(* CODESYS project Project1.project

Project tree, tasks and I/O mapping:
  PLC_AC500_V3 : PM5032-T-ETH, ABB AG, order no. 1SAP123400R0x72, version 3.7.0.0
    application Application
      task Task (cyclic, interval t#10ms, priority 14, watchdog t#20ms x 1) calls batching8, batching7
      task VISU_TASK (cyclic, interval 100 ms, priority 16) calls VisuElems.Visu_Prg
      CheckConfigurationObject
      program PLC_PRG [ST]
      program batching1 [ST]
      Diagnosis/
        text list Diag_IO_Bus
        text list Diag_V3_PLC
      program batching2 [ST]
      program batching3 [ST]
      program batching4 [ST]
      visualisation batching4_vis
      program batching5 [ST]
      global variables GVL
      function block Auto_Batching [ST]
      function block Manual_Batching [ST]
      program batching6 [ST]
      function block Auto_Batching_V7 [ST]
      function block Manual_Batching_V7 [ST]
      program batching7 [ST]
      function block Auto_Batching_V8 [ST]
      function block Manual_Batching_V8 [ST]
      program batching8 [ST]
      function block Auto_Batching_V9 [ST]
      function block Manual_Batching_V9 [ST]
      program batching9 [ST]
    OnBoard_IO : 12DI/8DO-T/2DC, ABB AG, version 3.7.0.0
        unmapped channels: Fast inputs DI0-DI3, Fast inputs DI4-DI7, Standard inputs DI8-DI11, Digital inputs - Transistor, Fast outputs DO0-DO3, Fast outputs DO4-DO7, Digital outputs - Transistor
    IO_Bus : I/O-Bus, ABB AG, version 3.7.0.0
    Interfaces : Interfaces, ABB AG, version 3.7.0.0
      OptionSlot_1
      OptionSlot_2
      Ethernet : Ethernet, ABB AG, version 3.7.0.0
        ETH1 : IP Settings, ABB AG, version 3.7.0.0
          NetConfig : NetConfig, ABB AG, version 3.7.0.0
        Protocols : Client Protocols, ABB AG, version 3.7.0.0
    OnBoard_RTC : OnBoard RTC, ABB AG, version 3.7.0.0
  text list GlobalTextList
*)

// PLC_AC500_V3/Application/GVL
{attribute 'qualified_only'}
VAR_GLOBAL
    Recipe_Weights : ARRAY[1..20] OF REAL := [
        50.0,   // Mat 1 (Auto Silo 1)
        15.0,   // Mat 2 (Auto Silo 2)
        28.0,   // Mat 3
        31.0,   // Mat 4 (Auto Silo 4)
        150.0,  // Mat 5 (Auto Silo 5)
        10.0,   // Mat 6 (Auto Silo 6)
        12.0,   // Mat 7 (Manual Silo 7)
        8.0,    // Mat 8 (Manual Silo 8)
        25.0,   // Mat 9 (Manual Silo 9)
        5.0,    // Mat 10 (Manual Silo 10)
        18.0,   // Mat 11 (Manual Silo 11)
        22.0,   // Mat 12 (Manual Silo 12)
        30.0,   // Mat 13 (Manual Silo 13)
        14.0,   // Mat 14 (Manual Silo 14)
        9.0,    // Mat 15 (Manual Silo 15)
        11.0,   // Mat 16 (Manual Silo 16)
        0.0, 0.0, 0.0, 0.0
    ];
END_VAR

// PLC_AC500_V3/Application/batching8
PROGRAM batching8
VAR
    Auto_Ctrl : Auto_Batching_V8;
    Manual_Ctrl : Manual_Batching_V8;
    
    (* Global Inputs & Toggles *)
    Start_Button : BOOL;
    E_Stop_Active : BOOL;
    
    (* Parallel Weight Feedbacks *)
    load_cell_auto : REAL;
    load_cell_manual : REAL;
    
    (* Sub-Block Diagnostic Indicators - Ordered exactly below loadcell *)
    Auto_Active_Mat : INT;
    Auto_Active_Bin : INT;
    Auto_Active_Target : REAL; // Active Target Weight for Auto (displays GVL setpoint)
    Auto_Err : INT;
    Auto_Msg : STRING;
    
    Manual_Active_Mat : INT;
    Manual_Active_Bin : INT;
    Manual_Active_Target : REAL; // Active Target Weight for Manual (displays GVL setpoint)
    Manual_Err : INT;
    Manual_Msg : STRING;
    
    (* Process Outputs *)
    Auto_Bin : ARRAY[1..6] OF BOOL; // Valve control outputs (Coarse)
    auto_bin_cutoff : ARRAY[1..6] OF BOOL; // Cutoff indicators (Fine)
    auto_bin_motor : ARRAY[1..6] OF BOOL; // Conveyor/feeder motor outputs
    
    Manual_Bin : ARRAY[1..10] OF BOOL; // Prompt indicators (Coarse)
    manual_bin_cutoff : ARRAY[1..10] OF BOOL; // Cutoff indicators (Fine)
    manual_bin_motor : ARRAY[1..10] OF BOOL; // Conveyor/feeder motor outputs
    
    Auto_Weights : ARRAY[1..6] OF REAL;
    Manual_Weights : ARRAY[1..10] OF REAL;
    
    Auto_Complete : BOOL;
    Manual_Complete : BOOL;
    Sequence_Complete : BOOL;
    
    (* Diagnostics & Interlocks *)
    Error_Code : INT := 0;
    Status_Message : STRING := 'System Ready';
    
    (* Array Configurations & Mapping - Renamed for clarity *)
    Auto_Bin_Material_Mapping : ARRAY[1..6] OF INT := [1, 2, 0, 4, 5, 6];
    Manual_Bin_Material_Mapping : ARRAY[1..10] OF INT := [7, 8, 0, 10, 11, 12, 13, 14, 15, 16];
    Auto_Bin_Cutoff_Weights : ARRAY[1..6] OF REAL := [2.0, 1.5, 0.0, 3.0, 5.0, 1.0]; // Cutoff margins (kg)
    Manual_Bin_Cutoff_Weights : ARRAY[1..10] OF REAL := [2.0, 1.5, 0.0, 3.0, 5.0, 1.0, 2.0, 2.0, 2.0, 2.0];
    
    i : INT;
    j : INT;
    Duplicate_Found : BOOL;
    Invalid_Material_Range : BOOL;
    Zero_Target_Found : BOOL;
    Conf_Err_Id : INT;
END_VAR

(* 1. STARTUP CONFIGURATION CHECKS *)
Duplicate_Found := FALSE;
Invalid_Material_Range := FALSE;
Zero_Target_Found := FALSE;

FOR i := 1 TO 6 DO
    (* Check 2: Out of Range (Auto) *)
    IF Auto_Bin_Material_Mapping[i] < 0 OR Auto_Bin_Material_Mapping[i] > 20 THEN
        Invalid_Material_Range := TRUE;
    END_IF;
    
    (* Check 3: Zero Target (Auto) *)
    IF Auto_Bin_Material_Mapping[i] <> 0 AND Auto_Bin_Material_Mapping[i] <= 20 THEN
        IF GVL.Recipe_Weights[Auto_Bin_Material_Mapping[i]] = 0.0 THEN
            Zero_Target_Found := TRUE;
        END_IF;
    END_IF;
    
    (* Check 1: Duplicate Cross-Array Material ID *)
    IF Auto_Bin_Material_Mapping[i] <> 0 AND Auto_Bin_Material_Mapping[i] <= 20 THEN
        FOR j := 1 TO 10 DO
            IF Auto_Bin_Material_Mapping[i] = Manual_Bin_Material_Mapping[j] THEN
                Duplicate_Found := TRUE;
            END_IF;
        END_FOR;
    END_IF;
END_FOR;

FOR j := 1 TO 10 DO
    (* Check 2: Out of Range (Manual) *)
    IF Manual_Bin_Material_Mapping[j] < 0 OR Manual_Bin_Material_Mapping[j] > 20 THEN
        Invalid_Material_Range := TRUE;
    END_IF;
    
    (* Check 3: Zero Target (Manual) *)
    IF Manual_Bin_Material_Mapping[j] <> 0 AND Manual_Bin_Material_Mapping[j] <= 20 THEN
        IF GVL.Recipe_Weights[Manual_Bin_Material_Mapping[j]] = 0.0 THEN
            Zero_Target_Found := TRUE;
        END_IF;
    END_IF;
END_FOR;

(* Configuration Error Resolution *)
IF Duplicate_Found THEN
    Error_Code := 1;
    Status_Message := 'Error 1: Duplicate Material ID mapped in Auto and Manual!';
ELSIF Invalid_Material_Range THEN
    Error_Code := 2;
    Status_Message := 'Error 2: Material Index configuration out of range (1..20)!';
ELSIF Zero_Target_Found THEN
    Error_Code := 3;
    Status_Message := 'Error 3: Configured Material ID has a 0.0 kg target weight!';
ELSE
    IF Error_Code <= 3 THEN
        Error_Code := 0;
    END_IF;
END_IF;

(* Abort sequences if a configuration error exists *)
IF Error_Code >= 1 AND Error_Code <= 3 THEN
    FOR i := 1 TO 6 DO Auto_Bin[i] := FALSE; auto_bin_cutoff[i] := FALSE; auto_bin_motor[i] := FALSE; END_FOR;
    FOR i := 1 TO 10 DO Manual_Bin[i] := FALSE; manual_bin_cutoff[i] := FALSE; manual_bin_motor[i] := FALSE; END_FOR;
    Auto_Ctrl(Start_Button := FALSE, E_Stop_Active := TRUE, load_cell_value := load_cell_auto);
    Manual_Ctrl(Start_Button := FALSE, E_Stop_Active := TRUE, load_cell_value := load_cell_manual);
    Auto_Active_Target := 0.0;
    Manual_Active_Target := 0.0;
    RETURN;
END_IF;


(* 2. CONCURRENT EXECUTION OF FB INSTANCES *)
Auto_Ctrl(
    Start_Button := Start_Button,
    E_Stop_Active := E_Stop_Active,
    load_cell_value := load_cell_auto,
    Auto_Bin_Material_Mapping := Auto_Bin_Material_Mapping,
    Auto_Bin_Cutoff_Weights := Auto_Bin_Cutoff_Weights,
    Auto_Bin => Auto_Bin,
    auto_bin_cutoff => auto_bin_cutoff,
    auto_bin_motor => auto_bin_motor,
    Actual_Weights => Auto_Weights,
    Sequence_Complete => Auto_Complete,
    Active_Material_ID => Auto_Active_Mat,
    Active_Bin_ID => Auto_Active_Bin,
    Active_Target_Weight => Auto_Active_Target,
    Error_Code => Auto_Err,
    Status_Message => Auto_Msg
);

Manual_Ctrl(
    Start_Button := Start_Button,
    E_Stop_Active := E_Stop_Active,
    load_cell_value := load_cell_manual,
    Manual_Bin_Material_Mapping := Manual_Bin_Material_Mapping,
    Manual_Bin_Cutoff_Weights := Manual_Bin_Cutoff_Weights,
    Manual_Bin => Manual_Bin,
    manual_bin_cutoff => manual_bin_cutoff,
    manual_bin_motor => manual_bin_motor,
    Actual_Weights => Manual_Weights,
    Sequence_Complete => Manual_Complete,
    Active_Material_ID => Manual_Active_Mat,
    Active_Bin_ID => Manual_Active_Bin,
    Active_Target_Weight => Manual_Active_Target,
    Error_Code => Manual_Err,
    Status_Message => Manual_Msg
);

(* Runtime Error Mapping & Aggregation *)
IF Auto_Err <> 0 THEN
    Error_Code := Auto_Err;
    Status_Message := CONCAT('Auto Error: ', Auto_Msg);
ELSIF Manual_Err <> 0 THEN
    Error_Code := Manual_Err;
    Status_Message := CONCAT('Manual Error: ', Manual_Msg);
ELSE
    Error_Code := 0;
    
    Sequence_Complete := Auto_Complete AND Manual_Complete;
    IF Sequence_Complete THEN
        Status_Message := 'Batch Sequence Completed';
    ELSIF Start_Button THEN
        Status_Message := 'Batch Sequence Running';
    ELSE
        Status_Message := 'System Ready';
    END_IF;
END_IF;

END_PROGRAM

// PLC_AC500_V3/Application/Auto_Batching_V8
FUNCTION_BLOCK Auto_Batching_V8
VAR_INPUT
    Start_Button : BOOL;      // Signal to start the batching sequence
    E_Stop_Active : BOOL;     // Emergency Stop active signal
    Discharge_Bin_Feedback : ARRAY[1..6] OF BOOL; // Physical valve feedbacks
    Auto_Bin_Material_Mapping : ARRAY[1..6] OF INT; // Material index mapping for 6 bins
    Auto_Bin_Cutoff_Weights : ARRAY[1..6] OF REAL; // Cutoff weight thresholds (kg)
END_VAR
VAR_IN_OUT
    load_cell_value : REAL;   // Weight value read/written from load cell
END_VAR
VAR_OUTPUT
    Auto_Bin : ARRAY[1..6] OF BOOL; // Coarse feed valve outputs
    auto_bin_cutoff : ARRAY[1..6] OF BOOL; // Fine feed cutoff trigger indicators
    auto_bin_motor : ARRAY[1..6] OF BOOL; // Main conveyor motor outputs
    Actual_Weights : ARRAY[1..6] OF REAL; // Actual weight poured per silo
    Sequence_Complete : BOOL;  // Batch complete flag
    Active_Material_ID : INT;  // Currently active ingredient ID
    Active_Bin_ID : INT;       // Currently active physical Bin ID (1..6)
    Active_Target_Weight : REAL; // Recipe target weight of active bin
    Error_Code : INT;          // Active error code
    Status_Message : STRING;   // Diagnostic text message
END_VAR
VAR
    Step : INT := 0;          // State machine index (0: Idle, 1..6: Bins, 11..16: Delays, 7: Settling, 8: Complete, 99: Error)
    bin_last_weight : REAL;   // Baseline weight on the load cell before starting current bin
    actual_bin : REAL;        // Current weight added from active bin
    target_act_bin : REAL;    // Target weight to add from the active bin
    bin_set_value : REAL;     // Setpoint weight for current active step
    cutoff_trigger_weight : REAL; // Calculated target threshold weight minus cutoff value
    
    Mat_Idx : INT;
    i : INT;                  // General loop index
    
    (* TIMERS FOR TRANSITIONS & DELAYS *)
    Transition_Timer : TON;
    Completion_Timer : TON;
    Step_Delay_Time : TIME := T#2S;
    Post_Complete_Delay : TIME := T#2S;
    
    (* SELF-CONTAINED SIMULATION VARIABLES *)
    Simulation_Mode : BOOL := TRUE;
    Sim_Rate : REAL := 10.0;            // Simulated pouring speed (10.0 kg/s)
    Sim_Timer : TON;
    Start_Sim_Weight : REAL;
    Discharge_Active : BOOL;
END_VAR

(* Auto Batching FB V8 matching batching7 sequence exactly *)

(* 1. SELF-CONTAINED SIMULATION WEIGHT MANAGEMENT *)
IF Simulation_Mode AND Step <> 99 THEN
    (* Reset simulation to baseline *)
    IF Step = 0 AND NOT Start_Button AND NOT Sequence_Complete THEN
        load_cell_value := 0.0;
        bin_last_weight := 0.0;
        Start_Sim_Weight := 0.0;
        Sim_Timer(IN := FALSE);
    END_IF;
    
    (* Check if any valve is actively discharging *)
    Discharge_Active := FALSE;
    IF Step >= 1 AND Step <= 6 THEN
        Discharge_Active := auto_bin_motor[Step];
    END_IF;
    
    (* Simulate weight gain on the load cell *)
    IF Discharge_Active THEN
        Sim_Timer(IN := TRUE, PT := T#1000S);
        load_cell_value := Start_Sim_Weight + (TIME_TO_REAL(Sim_Timer.ET) / 1000.0) * Sim_Rate;
    ELSE
        Sim_Timer(IN := FALSE);
        Start_Sim_Weight := load_cell_value;
    END_IF;
END_IF;


(* 2. EMERGENCY STOP LOGIC (Error 12) *)
IF E_Stop_Active THEN
    FOR i := 1 TO 6 DO
        Auto_Bin[i] := FALSE;
        auto_bin_cutoff[i] := FALSE;
        auto_bin_motor[i] := FALSE;
    END_FOR;
    Sequence_Complete := FALSE;
    Active_Material_ID := 0;
    Active_Bin_ID := 0;
    Active_Target_Weight := 0.0;
    Error_Code := 12;
    Status_Message := 'Error 12: Emergency Stop Active!';
    Step := 99;
    Transition_Timer(IN := FALSE);
    Completion_Timer(IN := FALSE);
    RETURN;
END_IF;


(* 3. RECIPE SEQUENCE START *)
IF Step = 0 AND Start_Button THEN
    Step := 1;
    bin_last_weight := load_cell_value;
    Sequence_Complete := FALSE;
    Error_Code := 0;
    Status_Message := 'Auto Batch Started';
    Active_Target_Weight := 0.0;
    (* Clear actual weights and outputs on start *)
    FOR i := 1 TO 6 DO
        Actual_Weights[i] := 0.0;
        Auto_Bin[i] := FALSE;
        auto_bin_cutoff[i] := FALSE;
        auto_bin_motor[i] := FALSE;
    END_FOR;
END_IF;


(* 4. SEQUENCE CONTROL STATE MACHINE *)
CASE Step OF
    0:
        Active_Material_ID := 0;
        Active_Bin_ID := 0;
        Active_Target_Weight := 0.0;
        IF Error_Code = 0 THEN Status_Message := 'Auto Idle'; END_IF;
        
    1..6: (* Discharging Silos 1 to 6 *)
        Mat_Idx := Auto_Bin_Material_Mapping[Step];
        
        IF Mat_Idx = 0 THEN
            (* Skip this bin instantly *)
            Step := Step + 1;
        ELSE
            (* Fetch target weight from global Recipe_Weights array *)
            bin_set_value := GVL.Recipe_Weights[Mat_Idx];
            target_act_bin := bin_set_value;
            Active_Target_Weight := target_act_bin;
            
            (* Calculate weight added by current active bin *)
            actual_bin := load_cell_value - bin_last_weight;
            Actual_Weights[Step] := actual_bin;
            
            (* Get cutoff threshold *)
            cutoff_trigger_weight := target_act_bin - Auto_Bin_Cutoff_Weights[Step];
            
            Active_Material_ID := Mat_Idx;
            Active_Bin_ID := Step;
            Status_Message := 'Auto Pouring';
            
            (* COARSE/FINE FEED TRANSITIONS *)
            IF actual_bin < cutoff_trigger_weight THEN
                (* Phase 1: Coarse Feed (Conveyor Motor ON, Main Valve ON, Fine Cutoff OFF) *)
                Auto_Bin[Step] := TRUE;
                auto_bin_cutoff[Step] := FALSE;
                auto_bin_motor[Step] := TRUE;
            ELSIF actual_bin < target_act_bin THEN
                (* Phase 2: Fine Feed (Conveyor Motor ON, Main Valve OFF, Fine Cutoff ON) *)
                Auto_Bin[Step] := FALSE;
                auto_bin_cutoff[Step] := TRUE;
                auto_bin_motor[Step] := TRUE;
            ELSE
                (* Phase 3: Completed (All OFF) *)
                Auto_Bin[Step] := FALSE;
                auto_bin_cutoff[Step] := FALSE;
                auto_bin_motor[Step] := FALSE;
                bin_last_weight := load_cell_value;
                Active_Target_Weight := 0.0;
                Step := 10 + Step; // Offset to separate transition states
            END_IF;
            
            (* RUNTIME CHECKS *)
            (* Check 21 & 22: Scale Limits *)
            IF load_cell_value > 500.0 THEN
                Error_Code := 21;
                Status_Message := 'Error 21: Scale Overloaded!';
                Step := 99;
                RETURN;
            ELSIF load_cell_value < 0.0 THEN
                Error_Code := 22;
                Status_Message := 'Error 22: Scale Underloaded/Fault!';
                Step := 99;
                RETURN;
            END_IF;
        END_IF;

    11..15: (* Transition Delays (Between Bins) *)
        Active_Material_ID := 0;
        Active_Bin_ID := 0;
        Active_Target_Weight := 0.0;
        Status_Message := 'Transition Delay';
        
        Transition_Timer(IN := TRUE, PT := Step_Delay_Time);
        IF Transition_Timer.Q THEN
            Transition_Timer(IN := FALSE);
            Step := (Step - 10) + 1; // Advance to next bin
        END_IF;
        
    16: (* Transition Delay After Last Bin (Bin 6) Closes *)
        Active_Material_ID := 0;
        Active_Bin_ID := 0;
        Active_Target_Weight := 0.0;
        Status_Message := 'Settling Last Bin';
        
        Transition_Timer(IN := TRUE, PT := Step_Delay_Time);
        IF Transition_Timer.Q THEN
            Transition_Timer(IN := FALSE);
            Step := 7; // Go to post-discharge wait step
        END_IF;

    7: (* Wait 2 Seconds After Closing the Last Bin *)
        Active_Material_ID := 0;
        Active_Bin_ID := 0;
        Active_Target_Weight := 0.0;
        Status_Message := 'Settling Delay';
        Completion_Timer(IN := TRUE, PT := Post_Complete_Delay);
        IF Completion_Timer.Q THEN
            Completion_Timer(IN := FALSE);
            Step := 8; // Proceed to reset last weight
        END_IF;
        
    8: (* Reset bin_last_weight to 0 & Complete *)
        Active_Material_ID := 0;
        Active_Bin_ID := 0;
        Active_Target_Weight := 0.0;
        Status_Message := 'Sequence Completed';
        bin_last_weight := 0.0;
        Sequence_Complete := TRUE;
        
        IF NOT Start_Button THEN
            Step := 0;
            Sequence_Complete := FALSE;
            (* Reset all actual weights at completion once start is released *)
            FOR i := 1 TO 6 DO
                Actual_Weights[i] := 0.0;
            END_FOR;
        END_IF;
        
    99: (* Error Abort state *)
        FOR i := 1 TO 6 DO 
            Auto_Bin[i] := FALSE; 
            auto_bin_cutoff[i] := FALSE;
            auto_bin_motor[i] := FALSE;
        END_FOR;
        Active_Material_ID := 0;
        Active_Bin_ID := 0;
        Active_Target_Weight := 0.0;
        IF NOT Start_Button THEN
            Step := 0;
            Error_Code := 0;
            Status_Message := 'Auto Idle';
        END_IF;
END_CASE;

END_FUNCTION_BLOCK

// PLC_AC500_V3/Application/batching7
PROGRAM batching7
VAR
    Auto_Ctrl : Auto_Batching_V7;
    Manual_Ctrl : Manual_Batching_V7;
    
    (* Global Inputs & Toggles *)
    Start_Button : BOOL;
    E_Stop_Active : BOOL;
    
    (* Parallel Weight Feedbacks *)
    load_cell_auto : REAL;
    load_cell_manual : REAL;
    
    (* Process Outputs *)
    Auto_Bin : ARRAY[1..6] OF BOOL;
    Manual_Bin : ARRAY[1..10] OF BOOL;
    
    Auto_Weights : ARRAY[1..6] OF REAL;
    Manual_Weights : ARRAY[1..10] OF REAL;
    
    Auto_Complete : BOOL;
    Manual_Complete : BOOL;
    Sequence_Complete : BOOL;
    
    (* Cross-Validation *)
    Error_Code : INT := 0; // 0 = OK, 1 = Duplicate Material ID detected
    Status_Message : STRING := 'System Ready';
    
    (* Arrays defined here to allow check before FB execution *)
    Bin_Material_Index : ARRAY[1..6] OF INT := [1, 2, 0, 4, 5, 6];
    Bin_Manual_Index : ARRAY[1..10] OF INT := [7, 8, 0, 10, 11, 12, 13, 14, 15, 16];
    
    (* Active IDs as integer monitors *)
    Auto_Active_Mat : INT;
    Auto_Active_Bin : INT;
    Manual_Active_Mat : INT;
    Manual_Active_Bin : INT;
    
    i : INT;
    j : INT;
    Duplicate_Found : BOOL;
END_VAR

(* 1. CROSS-ARRAY DISTINCT MATERIAL VALIDATION *)
Duplicate_Found := FALSE;
FOR i := 1 TO 6 DO
    IF Bin_Material_Index[i] <> 0 THEN
        FOR j := 1 TO 10 DO
            IF Bin_Material_Index[i] = Bin_Manual_Index[j] THEN
                Duplicate_Found := TRUE;
            END_IF;
        END_FOR;
    END_IF;
END_FOR;

IF Duplicate_Found THEN
    Error_Code := 1;
    Status_Message := 'Error 1: Duplicate Material ID in Auto and Manual tables!';
    
    (* Shut off all outputs and abort execution *)
    FOR i := 1 TO 6 DO Auto_Bin[i] := FALSE; END_FOR;
    FOR i := 1 TO 10 DO Manual_Bin[i] := FALSE; END_FOR;
    
    (* Reset control blocks *)
    Auto_Ctrl(Start_Button := FALSE, E_Stop_Active := TRUE);
    Manual_Ctrl(Start_Button := FALSE, E_Stop_Active := TRUE);
    RETURN;
ELSE
    Error_Code := 0;
END_IF;

(* 2. EXECUTION OF BATCH CONTROLLERS *)
Auto_Ctrl(
    Start_Button := Start_Button,
    E_Stop_Active := E_Stop_Active,
    load_cell_value := load_cell_auto,
    Bin_Material_Index := Bin_Material_Index,
    Auto_Bin => Auto_Bin,
    Actual_Weights => Auto_Weights,
    Sequence_Complete => Auto_Complete,
    Active_Material_ID => Auto_Active_Mat,
    Active_Bin_ID => Auto_Active_Bin
);

Manual_Ctrl(
    Start_Button := Start_Button,
    E_Stop_Active := E_Stop_Active,
    load_cell_value := load_cell_manual,
    Bin_Manual_Index := Bin_Manual_Index,
    Manual_Bin => Manual_Bin,
    Actual_Weights => Manual_Weights,
    Sequence_Complete => Manual_Complete,
    Active_Material_ID => Manual_Active_Mat,
    Active_Bin_ID => Manual_Active_Bin
);

Sequence_Complete := Auto_Complete AND Manual_Complete;

IF Sequence_Complete THEN
    Status_Message := 'Batch Completed';
ELSIF Start_Button THEN
    Status_Message := 'Batch In Progress';
ELSE
    Status_Message := 'System Ready';
END_IF;

END_PROGRAM

// PLC_AC500_V3/Application/Auto_Batching_V7
FUNCTION_BLOCK Auto_Batching_V7
VAR_INPUT
    Start_Button : BOOL;      // Signal to start the batching sequence
    E_Stop_Active : BOOL;     // Emergency Stop active signal
    load_cell_value : REAL;   // Weight value read from load cell
    Discharge_Bin_Feedback : ARRAY[1..6] OF BOOL; // Physical valve feedbacks
    Bin_Material_Index : ARRAY[1..6] OF INT;      // Mapped material index inputs
END_VAR
VAR_OUTPUT
    Auto_Bin : ARRAY[1..6] OF BOOL; // Motor/valve control outputs
    Actual_Weights : ARRAY[1..6] OF REAL; // Actual weight poured per silo
    Sequence_Complete : BOOL;  // Batch complete flag
    Active_Material_ID : INT;  // Currently active ingredient ID
    Active_Bin_ID : INT;       // Currently active physical Bin ID (1..6)
END_VAR
VAR
    Step : INT := 0;          // State machine index (0: Idle, 1..6: Bins, 7: Delay, 8: Reset)
    bin_last_weight : REAL;   // Baseline weight on the load cell before starting current bin
    actual_bin : REAL;        // Current weight added from active bin
    target_act_bin : REAL;    // Target weight to add from the active bin
    bin_set_value : REAL;     // Setpoint weight for current active step
    
    Mat_Idx : INT;
    i : INT;                  // General loop index
    
    (* TIMERS FOR TRANSITIONS & DELAYS *)
    Transition_Timer : TON;
    Completion_Timer : TON;
    Step_Delay_Time : TIME := T#2S;
    Post_Complete_Delay : TIME := T#2S;
    
    (* SELF-CONTAINED SIMULATION VARIABLES *)
    Simulation_Mode : BOOL := TRUE;
    Sim_Rate : REAL := 10.0;            // Simulated pouring speed (10.0 kg/s)
    Sim_Timer : TON;
    Start_Sim_Weight : REAL;
    Discharge_Active : BOOL;
END_VAR

(* Cumulative Gain-in-Weight Auto Batching FB V7 *)

(* 1. SELF-CONTAINED SIMULATION WEIGHT MANAGEMENT *)
IF Simulation_Mode THEN
    (* Reset simulation to baseline (e.g. 2.0 kg) *)
    IF Step = 0 AND NOT Start_Button AND NOT Sequence_Complete THEN
        load_cell_value := 2.0;
        bin_last_weight := 2.0;
        Start_Sim_Weight := 2.0;
        Sim_Timer(IN := FALSE);
    END_IF;
    
    (* Check if any valve is actively discharging *)
    Discharge_Active := FALSE;
    IF Step >= 1 AND Step <= 6 THEN
        Discharge_Active := Auto_Bin[Step];
    END_IF;
    
    (* Simulate weight gain on the load cell *)
    IF Discharge_Active THEN
        Sim_Timer(IN := TRUE, PT := T#1000S);
        load_cell_value := Start_Sim_Weight + (TIME_TO_REAL(Sim_Timer.ET) / 1000.0) * Sim_Rate;
    ELSE
        Sim_Timer(IN := FALSE);
        Start_Sim_Weight := load_cell_value;
    END_IF;
END_IF;


(* 2. EMERGENCY STOP LOGIC *)
IF E_Stop_Active THEN
    FOR i := 1 TO 6 DO
        Auto_Bin[i] := FALSE;
        Actual_Weights[i] := 0.0;
    END_FOR;
    Sequence_Complete := FALSE;
    Step := 0;
    Active_Material_ID := 0;
    Active_Bin_ID := 0;
    Transition_Timer(IN := FALSE);
    Completion_Timer(IN := FALSE);
    RETURN;
END_IF;


(* 3. RECIPE SEQUENCE START *)
IF Step = 0 AND Start_Button THEN
    Step := 1;
    bin_last_weight := load_cell_value;
    Sequence_Complete := FALSE;
    (* Clear actual weights on start *)
    FOR i := 1 TO 6 DO
        Actual_Weights[i] := 0.0;
    END_FOR;
END_IF;


(* 4. SEQUENCE CONTROL STATE MACHINE *)
CASE Step OF
    0:
        Active_Material_ID := 0;
        Active_Bin_ID := 0;
        
    1..6: (* Discharging Silos 1 to 6 *)
        Mat_Idx := Bin_Material_Index[Step];
        
        IF Mat_Idx = 0 THEN
            (* Skip this bin instantly *)
            Step := Step + 1;
        ELSE
            (* Fetch target weight from global Recipe_Weights array *)
            bin_set_value := GVL.Recipe_Weights[Mat_Idx];
            target_act_bin := bin_set_value;
            
            (* Calculate weight added by current active bin *)
            actual_bin := load_cell_value - bin_last_weight;
            
            (* Update the actual weight in the array for the active bin *)
            Actual_Weights[Step] := actual_bin;
            
            (* Open discharge output valve *)
            Auto_Bin[Step] := TRUE;
            
            (* Output currently active IDs *)
            Active_Material_ID := Mat_Idx;
            Active_Bin_ID := Step;
            
            (* Check if target weight has been achieved *)
            IF actual_bin >= target_act_bin THEN
                Auto_Bin[Step] := FALSE;
                
                (* Set new baseline for the next step *)
                bin_last_weight := load_cell_value;
                
                (* Go to transition delay *)
                Step := 10 + Step; // Offset to separate transition states
            END_IF;
        END_IF;

    11..15: (* Transition Delays (Between Bins) *)
        Active_Material_ID := 0;
        Active_Bin_ID := 0;
        Transition_Timer(IN := TRUE, PT := Step_Delay_Time);
        IF Transition_Timer.Q AND (NOT Auto_Bin[Step - 10] OR NOT Discharge_Bin_Feedback[Step - 10]) THEN
            Transition_Timer(IN := FALSE);
            Step := (Step - 10) + 1; // Advance to next bin
        END_IF;
        
    16: (* Transition Delay After Last Bin (Bin 6) Closes *)
        Active_Material_ID := 0;
        Active_Bin_ID := 0;
        Transition_Timer(IN := TRUE, PT := Step_Delay_Time);
        IF Transition_Timer.Q AND (NOT Auto_Bin[6] OR NOT Discharge_Bin_Feedback[6]) THEN
            Transition_Timer(IN := FALSE);
            Step := 7; // Go to post-discharge wait step
        END_IF;

    7: (* Wait 2 Seconds After Closing the Last Bin *)
        Active_Material_ID := 0;
        Active_Bin_ID := 0;
        Completion_Timer(IN := TRUE, PT := Post_Complete_Delay);
        IF Completion_Timer.Q THEN
            Completion_Timer(IN := FALSE);
            Step := 8; // Proceed to reset last weight
        END_IF;
        
    8: (* Reset bin_last_weight to 0 & Complete *)
        Active_Material_ID := 0;
        Active_Bin_ID := 0;
        bin_last_weight := 0.0;
        Sequence_Complete := TRUE;
        
        IF NOT Start_Button THEN
            Step := 0;
            Sequence_Complete := FALSE;
            (* Reset all actual weights at completion once start is released *)
            FOR i := 1 TO 6 DO
                Actual_Weights[i] := 0.0;
            END_FOR;
        END_IF;
END_CASE;

END_FUNCTION_BLOCK

// PLC_AC500_V3/Application/Manual_Batching_V7
FUNCTION_BLOCK Manual_Batching_V7
VAR_INPUT
    Start_Button : BOOL;      // Signal to start the batching sequence
    E_Stop_Active : BOOL;     // Emergency Stop active signal
    load_cell_value : REAL;   // Weight value read from load cell
    Bin_Manual_Index : ARRAY[1..10] OF INT; // Mapped material index inputs
END_VAR
VAR_OUTPUT
    Manual_Bin : ARRAY[1..10] OF BOOL; // Prompts/indicators for Bins 7..16
    Actual_Weights : ARRAY[1..10] OF REAL; // Actual weight poured per silo
    Sequence_Complete : BOOL;  // Batch complete flag
    Active_Material_ID : INT;  // Currently active ingredient ID
    Active_Bin_ID : INT;       // Currently active physical Bin ID (7..16)
END_VAR
VAR
    Step : INT := 0;          // State machine index (0: Idle, 1..10: Bins, 11..20: Delays, 30: Settling, 40: Complete)
    bin_last_weight : REAL;   // Baseline weight on the load cell before starting current bin
    actual_bin : REAL;        // Current weight added from active bin
    target_act_bin : REAL;    // Target weight to add from the active bin
    bin_set_value : REAL;     // Setpoint weight for current active step
    
    Mat_Idx : INT;
    i : INT;                  // General loop index
    
    (* TIMERS FOR TRANSITIONS & DELAYS *)
    Transition_Timer : TON;
    Completion_Timer : TON;
    Step_Delay_Time : TIME := T#2S;
    Post_Complete_Delay : TIME := T#2S;
    
    (* SELF-CONTAINED SIMULATION VARIABLES *)
    Simulation_Mode : BOOL := TRUE;
    Sim_Rate : REAL := 10.0;            // Simulated pouring speed (10.0 kg/s)
    Sim_Timer : TON;
    Start_Sim_Weight : REAL;
    Discharge_Active : BOOL;
END_VAR

(* Cumulative Gain-in-Weight Manual Batching FB V7 *)

(* 1. SIMULATION WEIGHT MANAGEMENT *)
IF Simulation_Mode THEN
    (* Reset simulation to baseline (e.g. 2.0 kg) *)
    IF Step = 0 AND NOT Start_Button AND NOT Sequence_Complete THEN
        load_cell_value := 2.0;
        bin_last_weight := 2.0;
        Start_Sim_Weight := 2.0;
        Sim_Timer(IN := FALSE);
    END_IF;
    
    (* Check if operator is actively pouring *)
    Discharge_Active := FALSE;
    IF Step >= 1 AND Step <= 10 THEN
        Discharge_Active := Manual_Bin[Step];
    END_IF;
    
    (* Simulate weight gain on the load cell *)
    IF Discharge_Active THEN
        Sim_Timer(IN := TRUE, PT := T#1000S);
        load_cell_value := Start_Sim_Weight + (TIME_TO_REAL(Sim_Timer.ET) / 1000.0) * Sim_Rate;
    ELSE
        Sim_Timer(IN := FALSE);
        Start_Sim_Weight := load_cell_value;
    END_IF;
END_IF;


(* 2. EMERGENCY STOP LOGIC *)
IF E_Stop_Active THEN
    FOR i := 1 TO 10 DO
        Manual_Bin[i] := FALSE;
        Actual_Weights[i] := 0.0;
    END_FOR;
    Sequence_Complete := FALSE;
    Step := 0;
    Active_Material_ID := 0;
    Active_Bin_ID := 0;
    Transition_Timer(IN := FALSE);
    Completion_Timer(IN := FALSE);
    RETURN;
END_IF;


(* 3. RECIPE SEQUENCE START *)
IF Step = 0 AND Start_Button THEN
    Step := 1;
    bin_last_weight := load_cell_value;
    Sequence_Complete := FALSE;
    (* Clear actual weights on start *)
    FOR i := 1 TO 10 DO
        Actual_Weights[i] := 0.0;
    END_FOR;
END_IF;


(* 4. SEQUENCE CONTROL STATE MACHINE *)
CASE Step OF
    0:
        Active_Material_ID := 0;
        Active_Bin_ID := 0;
        
    1..10: (* Prompts Silos 7 to 16 *)
        Mat_Idx := Bin_Manual_Index[Step];
        
        IF Mat_Idx = 0 THEN
            (* Skip this bin instantly *)
            Step := Step + 1;
        ELSE
            (* Fetch target weight from global Recipe_Weights array *)
            bin_set_value := GVL.Recipe_Weights[Mat_Idx];
            target_act_bin := bin_set_value;
            
            (* Calculate weight added by current active bin *)
            actual_bin := load_cell_value - bin_last_weight;
            
            (* Update the actual weight in the array for the active bin *)
            Actual_Weights[Step] := actual_bin;
            
            (* Prompt operator indicator active *)
            Manual_Bin[Step] := TRUE;
            
            (* Output currently active IDs (Shift to physical Silo ID 7..16) *)
            Active_Material_ID := Mat_Idx;
            Active_Bin_ID := Step + 6;
            
            (* Check if target weight has been achieved *)
            IF actual_bin >= target_act_bin THEN
                Manual_Bin[Step] := FALSE;
                
                (* Set new baseline for the next step *)
                bin_last_weight := load_cell_value;
                
                (* Go to transition delay *)
                Step := 10 + Step; // Offset to separate transition states
            END_IF;
        END_IF;

    11..19: (* Transition Delays (Between Bins) *)
        Active_Material_ID := 0;
        Active_Bin_ID := 0;
        Transition_Timer(IN := TRUE, PT := Step_Delay_Time);
        IF Transition_Timer.Q THEN
            Transition_Timer(IN := FALSE);
            Step := (Step - 10) + 1; // Advance to next bin
        END_IF;
        
    20: (* Transition Delay After Last Bin (Bin 10) Closes *)
        Active_Material_ID := 0;
        Active_Bin_ID := 0;
        Transition_Timer(IN := TRUE, PT := Step_Delay_Time);
        IF Transition_Timer.Q THEN
            Transition_Timer(IN := FALSE);
            Step := 30; // Go to post-discharge wait step (State 30)
        END_IF;

    30: (* Wait 2 Seconds After Closing the Last Bin *)
        Active_Material_ID := 0;
        Active_Bin_ID := 0;
        Completion_Timer(IN := TRUE, PT := Post_Complete_Delay);
        IF Completion_Timer.Q THEN
            Completion_Timer(IN := FALSE);
            Step := 40; // Proceed to reset last weight (State 40)
        END_IF;
        
    40: (* Reset bin_last_weight to 0 & Complete *)
        Active_Material_ID := 0;
        Active_Bin_ID := 0;
        bin_last_weight := 0.0;
        Sequence_Complete := TRUE;
        
        IF NOT Start_Button THEN
            Step := 0;
            Sequence_Complete := FALSE;
            (* Reset all actual weights at completion once start is released *)
            FOR i := 1 TO 10 DO
                Actual_Weights[i] := 0.0;
            END_FOR;
        END_IF;
END_CASE;

END_FUNCTION_BLOCK

// PLC_AC500_V3/Application/Manual_Batching_V8
FUNCTION_BLOCK Manual_Batching_V8
VAR_INPUT
    Start_Button : BOOL;      // Signal to start the batching sequence
    E_Stop_Active : BOOL;     // Emergency Stop active signal
    Manual_Bin_Material_Mapping : ARRAY[1..10] OF INT; // Material index mapping for 10 manual silos
    Manual_Bin_Cutoff_Weights : ARRAY[1..10] OF REAL; // Cutoff weight thresholds (kg)
END_VAR
VAR_IN_OUT
    load_cell_value : REAL;   // Weight value read/written from load cell
END_VAR
VAR_OUTPUT
    Manual_Bin : ARRAY[1..10] OF BOOL; // Prompts/indicators for Bins 7..16
    manual_bin_cutoff : ARRAY[1..10] OF BOOL; // Manual pre-cutoff indicators
    manual_bin_motor : ARRAY[1..10] OF BOOL; // Main manual feeder motor outputs
    Actual_Weights : ARRAY[1..10] OF REAL; // Actual weight poured per silo
    Sequence_Complete : BOOL;  // Batch complete flag
    Active_Material_ID : INT;  // Currently active ingredient ID
    Active_Bin_ID : INT;       // Currently active physical Bin ID (7..16)
    Active_Target_Weight : REAL; // Recipe target weight of active bin
    Error_Code : INT;          // Active error code
    Status_Message : STRING;   // Diagnostic text message
END_VAR
VAR
    Step : INT := 0;          // State machine index (0: Idle, 1..10: Bins, 11..20: Delays, 30: Settling, 40: Complete, 99: Error)
    bin_last_weight : REAL;   // Baseline weight on the load cell before starting current bin
    actual_bin : REAL;        // Current weight added from active bin
    target_act_bin : REAL;    // Target weight to add from the active bin
    bin_set_value : REAL;     // Setpoint weight for current active step
    cutoff_trigger_weight : REAL; // Calculated target threshold weight minus cutoff value
    
    Mat_Idx : INT;
    i : INT;                  // General loop index
    
    (* TIMERS FOR TRANSITIONS & DELAYS *)
    Transition_Timer : TON;
    Completion_Timer : TON;
    Step_Delay_Time : TIME := T#2S;
    Post_Complete_Delay : TIME := T#2S;
    
    (* DIAGNOSTIC TIMERS *)
    Operator_Timer : TON;
    
    (* SELF-CONTAINED SIMULATION VARIABLES *)
    Simulation_Mode : BOOL := TRUE;
    Sim_Rate : REAL := 10.0;            // Simulated pouring speed (10.0 kg/s)
    Sim_Timer : TON;
    Start_Sim_Weight : REAL;
    Discharge_Active : BOOL;
END_VAR

(* Manual Batching FB V8 with Diagnostic Error Checks *)

(* 1. SIMULATION WEIGHT MANAGEMENT *)
IF Simulation_Mode AND Step <> 99 THEN
    (* Reset simulation to baseline *)
    IF Step = 0 AND NOT Start_Button AND NOT Sequence_Complete THEN
        load_cell_value := 0.0;
        bin_last_weight := 0.0;
        Start_Sim_Weight := 0.0;
        Sim_Timer(IN := FALSE);
    END_IF;
    
    (* Check if operator is actively pouring *)
    Discharge_Active := FALSE;
    IF Step >= 1 AND Step <= 10 THEN
        Discharge_Active := manual_bin_motor[Step];
    END_IF;
    
    (* Simulate weight gain on the load cell *)
    IF Discharge_Active THEN
        Sim_Timer(IN := TRUE, PT := T#1000S);
        load_cell_value := Start_Sim_Weight + (TIME_TO_REAL(Sim_Timer.ET) / 1000.0) * Sim_Rate;
    ELSE
        Sim_Timer(IN := FALSE);
        Start_Sim_Weight := load_cell_value;
    END_IF;
END_IF;


(* 2. EMERGENCY STOP LOGIC (Error 12) *)
IF E_Stop_Active THEN
    FOR i := 1 TO 10 DO
        Manual_Bin[i] := FALSE;
        manual_bin_cutoff[i] := FALSE;
        manual_bin_motor[i] := FALSE;
    END_FOR;
    Sequence_Complete := FALSE;
    Active_Material_ID := 0;
    Active_Bin_ID := 0;
    Active_Target_Weight := 0.0;
    Error_Code := 12;
    Status_Message := 'Error 12: Emergency Stop Active!';
    Step := 99;
    Transition_Timer(IN := FALSE);
    Completion_Timer(IN := FALSE);
    RETURN;
END_IF;


(* 3. RECIPE SEQUENCE START *)
IF Step = 0 AND Start_Button THEN
    Step := 1;
    bin_last_weight := load_cell_value;
    Sequence_Complete := FALSE;
    Error_Code := 0;
    Status_Message := 'Manual Batch Started';
    Active_Target_Weight := 0.0;
    (* Clear actual weights on start *)
    FOR i := 1 TO 10 DO
        Actual_Weights[i] := 0.0;
        Manual_Bin[i] := FALSE;
        manual_bin_cutoff[i] := FALSE;
        manual_bin_motor[i] := FALSE;
    END_FOR;
END_IF;


(* 4. SEQUENCE CONTROL STATE MACHINE *)
CASE Step OF
    0:
        Active_Material_ID := 0;
        Active_Bin_ID := 0;
        Active_Target_Weight := 0.0;
        IF Error_Code = 0 THEN Status_Message := 'Manual Idle'; END_IF;
        
    1..10: (* Prompts Silos 7 to 16 *)
        Mat_Idx := Manual_Bin_Material_Mapping[Step];
        
        IF Mat_Idx = 0 THEN
            (* Skip this bin instantly *)
            Step := Step + 1;
        ELSE
            (* Fetch target weight from global Recipe_Weights array *)
            bin_set_value := GVL.Recipe_Weights[Mat_Idx];
            target_act_bin := bin_set_value;
            Active_Target_Weight := target_act_bin;
            
            (* Calculate weight added by current active bin *)
            actual_bin := load_cell_value - bin_last_weight;
            Actual_Weights[Step] := actual_bin;
            
            (* Get cutoff threshold *)
            cutoff_trigger_weight := target_act_bin - Manual_Bin_Cutoff_Weights[Step];
            
            Active_Material_ID := Mat_Idx;
            Active_Bin_ID := Step + 6;
            Status_Message := 'Manual Pouring Active';
            
            (* COARSE/FINE FEED TRANSITIONS *)
            IF actual_bin < cutoff_trigger_weight THEN
                (* Phase 1: Coarse Feed (Motor ON, Prompt ON, Cutoff OFF) *)
                Manual_Bin[Step] := TRUE;
                manual_bin_cutoff[Step] := FALSE;
                manual_bin_motor[Step] := TRUE;
            ELSIF actual_bin < target_act_bin THEN
                (* Phase 2: Fine Feed (Motor ON, Prompt OFF, Cutoff ON) *)
                Manual_Bin[Step] := FALSE;
                manual_bin_cutoff[Step] := TRUE;
                manual_bin_motor[Step] := TRUE;
            ELSE
                (* Phase 3: Completed (All OFF) *)
                Manual_Bin[Step] := FALSE;
                manual_bin_cutoff[Step] := FALSE;
                manual_bin_motor[Step] := FALSE;
                bin_last_weight := load_cell_value;
                Active_Target_Weight := 0.0;
                Step := 10 + Step; // Offset to separate transition states
            END_IF;
            
            (* RUNTIME CHECKS *)
            (* Check 21 & 22: Scale Limits *)
            IF load_cell_value > 500.0 THEN
                Error_Code := 21;
                Status_Message := 'Error 21: Scale Overloaded!';
                Step := 99;
                RETURN;
            ELSIF load_cell_value < 0.0 THEN
                Error_Code := 22;
                Status_Message := 'Error 22: Scale Underloaded/Fault!';
                Step := 99;
                RETURN;
            END_IF;
            
            (* Check 30: Operator Timeout *)
            Operator_Timer(IN := manual_bin_motor[Step], PT := T#300S);
            IF Operator_Timer.Q THEN
                Error_Code := 30;
                Status_Message := 'Error 30: Manual Operator Timeout!';
                Step := 99;
                RETURN;
            END_IF;
        END_IF;

    11..19: (* Transition Delays (Between Bins) *)
        Active_Material_ID := 0;
        Active_Bin_ID := 0;
        Active_Target_Weight := 0.0;
        Status_Message := 'Transition Delay';
        Transition_Timer(IN := TRUE, PT := Step_Delay_Time);
        IF Transition_Timer.Q THEN
            Transition_Timer(IN := FALSE);
            Step := (Step - 10) + 1; // Advance to next bin
        END_IF;
        
    20: (* Transition Delay After Last Bin (Bin 10) Closes *)
        Active_Material_ID := 0;
        Active_Bin_ID := 0;
        Active_Target_Weight := 0.0;
        Status_Message := 'Settling Last Bin';
        Transition_Timer(IN := TRUE, PT := Step_Delay_Time);
        IF Transition_Timer.Q THEN
            Transition_Timer(IN := FALSE);
            Step := 30; // Go to post-discharge wait step (State 30)
        END_IF;

    30: (* Wait 2 Seconds After Closing the Last Bin *)
        Active_Material_ID := 0;
        Active_Bin_ID := 0;
        Active_Target_Weight := 0.0;
        Status_Message := 'Settling Delay';
        Completion_Timer(IN := TRUE, PT := Post_Complete_Delay);
        IF Completion_Timer.Q THEN
            Completion_Timer(IN := FALSE);
            Step := 40; // Proceed to reset last weight (State 40)
        END_IF;
        
    40: (* Reset bin_last_weight to 0 & Complete *)
        Active_Material_ID := 0;
        Active_Bin_ID := 0;
        Active_Target_Weight := 0.0;
        Status_Message := 'Sequence Completed';
        bin_last_weight := 0.0;
        Sequence_Complete := TRUE;
        
        IF NOT Start_Button THEN
            Step := 0;
            Sequence_Complete := FALSE;
            (* Reset all actual weights at completion once start is released *)
            FOR i := 1 TO 10 DO
                Actual_Weights[i] := 0.0;
            END_FOR;
        END_IF;
        
    99: (* Error Abort state *)
        FOR i := 1 TO 10 DO 
            Manual_Bin[i] := FALSE;
            manual_bin_cutoff[i] := FALSE;
            manual_bin_motor[i] := FALSE;
        END_FOR;
        Active_Material_ID := 0;
        Active_Bin_ID := 0;
        Active_Target_Weight := 0.0;
        IF NOT Start_Button THEN
            Step := 0;
            Error_Code := 0;
            Status_Message := 'Manual Idle';
        END_IF;
END_CASE;

END_FUNCTION_BLOCK

// PLC_AC500_V3/Application/PLC_PRG
PROGRAM PLC_PRG
VAR
END_VAR

END_PROGRAM

// PLC_AC500_V3/Application/batching1
PROGRAM batching1
VAR
    Step : INT := 0;
    
    (* Mode Control *)
    Auto_Mode : BOOL := TRUE; // TRUE for Auto, FALSE for Manual
    
    (* Control Buttons *)
    Start_Button : BOOL;      // Start button for Auto sequence
    E_Stop_Active : BOOL;     // Emergency Stop active signal (normally open logic in software)
    
    (* Manual Buttons *)
    Manual_Bin1 : BOOL;       // Manual discharge trigger for Bin 1
    Manual_Bin2 : BOOL;       // Manual discharge trigger for Bin 2
    Manual_Bin3 : BOOL;       // Manual discharge trigger for Bin 3
    
    (* Discharge outputs *)
    Discharge_Bin1 : BOOL;
    Discharge_Bin2 : BOOL;
    Discharge_Bin3 : BOOL;
    
    (* Valve feedback (set to TRUE when open, FALSE when closed) *)
    Discharge_Bin1_Feedback : BOOL;
    Discharge_Bin2_Feedback : BOOL;
    Discharge_Bin3_Feedback : BOOL;
    
    (* Empty status / feedback *)
    Bin1_Empty : BOOL;
    Bin2_Empty : BOOL;
    Bin3_Empty : BOOL;
    
    (* Weight sensors (optional feedback) *)
    Bin1_Weight : REAL;
    Bin2_Weight : REAL;
    Bin3_Weight : REAL;
    
    Sequence_Complete : BOOL;
    
    (* DELAYS FOR VISUAL MONITORING *)
    Bin3_Timer : TON;         // Timer for Bin 3 discharge
    Bin2_Timer : TON;         // Timer for Bin 2 discharge
    Bin1_Timer : TON;         // Timer for Bin 1 discharge
    Transition_Timer : TON;   // Timer for transitions between stages
    
    Min_Discharge_Time : TIME := T#3S;  // Minimum time each bin stays open to allow visibility (e.g. 3 seconds)
    Step_Delay_Time : TIME := T#2S;     // Wait time between closing one bin and opening the next (e.g. 2 seconds)
END_VAR

(* Discharging Sequence with Auto/Manual Mode, E-Stop, Manual Controls, and Monitoring Delays *)

(* Emergency Stop Logic - High Priority *)
IF E_Stop_Active THEN
    Discharge_Bin1 := FALSE;
    Discharge_Bin2 := FALSE;
    Discharge_Bin3 := FALSE;
    Sequence_Complete := FALSE;
    Step := 0;
    
    (* Reset Timers *)
    Bin3_Timer(IN := FALSE);
    Bin2_Timer(IN := FALSE);
    Bin1_Timer(IN := FALSE);
    Transition_Timer(IN := FALSE);
    RETURN; // Halt execution of the rest of the POU
END_IF;

(* Mode Selection *)
IF Auto_Mode THEN
    (* ================= AUTOMATIC MODE ================= *)
    CASE Step OF
        0: (* Idle state *)
            Discharge_Bin1 := FALSE;
            Discharge_Bin2 := FALSE;
            Discharge_Bin3 := FALSE;
            Sequence_Complete := FALSE;
            
            Bin3_Timer(IN := FALSE);
            Bin2_Timer(IN := FALSE);
            Bin1_Timer(IN := FALSE);
            Transition_Timer(IN := FALSE);
            
            IF Start_Button THEN
                Step := 10;
            END_IF
            
        10: (* Discharge Bin 3 - ON *)
            Discharge_Bin3 := TRUE;
            Discharge_Bin2 := FALSE;
            Discharge_Bin1 := FALSE;
            
            (* Run timer to ensure discharge is visible *)
            Bin3_Timer(IN := TRUE, PT := Min_Discharge_Time);
            
            (* Transition when empty AND minimum time has elapsed *)
            IF (Bin3_Empty OR Bin3_Weight <= 0) AND Bin3_Timer.Q THEN
                Bin3_Timer(IN := FALSE); // Reset timer
                Step := 15;
            END_IF
            
        15: (* Discharge Bin 3 - OFF & Wait Transition Delay *)
            Discharge_Bin3 := FALSE;
            Transition_Timer(IN := TRUE, PT := Step_Delay_Time);
            
            IF Transition_Timer.Q AND (NOT Discharge_Bin3_Feedback OR NOT Discharge_Bin3) THEN
                Transition_Timer(IN := FALSE); // Reset timer
                Step := 20;
            END_IF
            
        20: (* Discharge Bin 2 - ON *)
            Discharge_Bin2 := TRUE;
            Discharge_Bin3 := FALSE;
            Discharge_Bin1 := FALSE;
            
            Bin2_Timer(IN := TRUE, PT := Min_Discharge_Time);
            
            IF (Bin2_Empty OR Bin2_Weight <= 0) AND Bin2_Timer.Q THEN
                Bin2_Timer(IN := FALSE);
                Step := 25;
            END_IF
            
        25: (* Discharge Bin 2 - OFF & Wait Transition Delay *)
            Discharge_Bin2 := FALSE;
            Transition_Timer(IN := TRUE, PT := Step_Delay_Time);
            
            IF Transition_Timer.Q AND (NOT Discharge_Bin2_Feedback OR NOT Discharge_Bin2) THEN
                Transition_Timer(IN := FALSE);
                Step := 30;
            END_IF
            
        30: (* Discharge Bin 1 - ON *)
            Discharge_Bin1 := TRUE;
            Discharge_Bin3 := FALSE;
            Discharge_Bin2 := FALSE;
            
            Bin1_Timer(IN := TRUE, PT := Min_Discharge_Time);
            
            IF (Bin1_Empty OR Bin1_Weight <= 0) AND Bin1_Timer.Q THEN
                Bin1_Timer(IN := FALSE);
                Step := 35;
            END_IF
            
        35: (* Discharge Bin 1 - OFF & Wait Transition Delay *)
            Discharge_Bin1 := FALSE;
            Transition_Timer(IN := TRUE, PT := Step_Delay_Time);
            
            IF Transition_Timer.Q AND (NOT Discharge_Bin1_Feedback OR NOT Discharge_Bin1) THEN
                Transition_Timer(IN := FALSE);
                Step := 40;
            END_IF
            
        40: (* Sequence Complete *)
            Sequence_Complete := TRUE;
            IF NOT Start_Button THEN
                Step := 0;
            END_IF
    END_CASE;

ELSE
    (* ================= MANUAL MODE ================= *)
    Step := 0;
    Sequence_Complete := FALSE;
    
    (* Reset all timers *)
    Bin3_Timer(IN := FALSE);
    Bin2_Timer(IN := FALSE);
    Bin1_Timer(IN := FALSE);
    Transition_Timer(IN := FALSE);
    
    (* Separate buttons for each bin with interlinking *)
    IF Manual_Bin3 THEN
        Discharge_Bin3 := TRUE;
        Discharge_Bin2 := FALSE;
        Discharge_Bin1 := FALSE;
    ELSIF Manual_Bin2 THEN
        Discharge_Bin3 := FALSE;
        Discharge_Bin2 := TRUE;
        Discharge_Bin1 := FALSE;
    ELSIF Manual_Bin1 THEN
        Discharge_Bin3 := FALSE;
        Discharge_Bin2 := FALSE;
        Discharge_Bin1 := TRUE;
    ELSE
        Discharge_Bin3 := FALSE;
        Discharge_Bin2 := FALSE;
        Discharge_Bin1 := FALSE;
    END_IF;
END_IF;

END_PROGRAM

// PLC_AC500_V3/Application/batching2
PROGRAM batching2
VAR
    Step : INT := 0;
    
    (* Mode Control *)
    Auto_Mode : BOOL := TRUE; // TRUE for Auto, FALSE for Manual
    Simulation_Mode : BOOL := TRUE; // Set to TRUE for software simulation, FALSE for physical hardware
    
    (* Control Buttons *)
    Start_Button : BOOL;      // Start button for Auto sequence
    E_Stop_Active : BOOL;     // Emergency Stop active signal
    
    (* Manual Buttons *)
    Manual_Bin1 : BOOL;       // Manual discharge trigger for Bin 1
    Manual_Bin2 : BOOL;       // Manual discharge trigger for Bin 2
    Manual_Bin3 : BOOL;       // Manual discharge trigger for Bin 3
    
    (* Discharge outputs *)
    Discharge_Bin1 : BOOL;
    Discharge_Bin2 : BOOL;
    Discharge_Bin3 : BOOL;
    
    (* Valve feedback *)
    Discharge_Bin1_Feedback : BOOL;
    Discharge_Bin2_Feedback : BOOL;
    Discharge_Bin3_Feedback : BOOL;
    
    (* Modbus Weight Inputs (Current Weight of the Bins) *)
    Current_Weight_Bin1 : REAL; // Current load cell reading for Bin 1 (Water)
    Current_Weight_Bin2 : REAL; // Current load cell reading for Bin 2 (Aggregate)
    Current_Weight_Bin3 : REAL; // Current load cell reading for Bin 3 (Cement)
    
    (* Starting Weights (Captured at start of process) *)
    Start_Weight_Bin1 : REAL;   // Weight snapshot of Bin 1 at start
    Start_Weight_Bin2 : REAL;   // Weight snapshot of Bin 2 at start
    Start_Weight_Bin3 : REAL;   // Weight snapshot of Bin 3 at start
    
    (* Target Discharge Threshold Amounts *)
    Target_Amount_Bin1 : REAL := 0.5;  // Amount of Water to discharge (e.g. 0.5 L)
    Target_Amount_Bin2 : REAL := 1.5;  // Amount of Aggregate to discharge (e.g. 1.5 kg)
    Target_Amount_Bin3 : REAL := 1.0;  // Amount of Cement to discharge (e.g. 1.0 kg)
    
    (* Calculated Cutoff Weights *)
    Cutoff_Weight_Bin1 : REAL;
    Cutoff_Weight_Bin2 : REAL;
    Cutoff_Weight_Bin3 : REAL;
    
    Sequence_Complete : BOOL;
    Transition_Timer : TON;
    Step_Delay_Time : TIME := T#2S;     // Delay between closing one valve and opening the next
    
    (* TIMERS FOR WEIGHT DECREMENT (EXACT 1.0 kg/s SIMULATION) *)
    Bin3_Timer : TON;         // Tracks elapsed open time of Bin 3
    Bin2_Timer : TON;         // Tracks elapsed open time of Bin 2
    Bin1_Timer : TON;         // Tracks elapsed open time of Bin 1
    
    (* SIMULATION DISCHARGE RATES (units per second) *)
    Sim_Rate_Bin1 : REAL := 1.0;        // Water loss rate: 1.0 L / second
    Sim_Rate_Bin2 : REAL := 1.0;        // Aggregate loss rate: 1.0 kg / second
    Sim_Rate_Bin3 : REAL := 1.0;        // Cement loss rate: 1.0 kg / second
    
    (* Modbus Master instances for each load cell (Commented out for compile-safety in simulation) *)
    (*
    Read_LC1 : COM_MODMAST;
    Read_LC2 : COM_MODMAST;
    Read_LC3 : COM_MODMAST;
    *)
    
    (* Modbus buffers (Commented out for compile-safety in simulation) *)
    (*
    LC1_Buffer : ARRAY[0..1] OF WORD;
    LC2_Buffer : ARRAY[0..1] OF WORD;
    LC3_Buffer : ARRAY[0..1] OF WORD;
    *)
END_VAR

(* Discharging Sequence with Auto/Manual Mode, E-Stop, Manual Controls, and Loss-in-Weight Threshold Cutoffs *)

(* 1. SIMULATION LOGIC (To run without physical Modbus hardware) *)
IF Simulation_Mode THEN
    (* Initialize weights to start values in Idle state *)
    IF Step = 0 AND NOT Start_Button AND NOT Sequence_Complete THEN
        Current_Weight_Bin3 := 70.0; // 70 kg Cement
        Current_Weight_Bin2 := 50.0; // 50 kg Aggregate
        Current_Weight_Bin1 := 80.0; // 80 L Water
    END_IF;
    
    (* Dynamically reduce weights based on elapsed time of active discharge (scan-time independent) *)
    IF Discharge_Bin3 THEN
        Bin3_Timer(IN := TRUE, PT := T#1000S);
        Current_Weight_Bin3 := Start_Weight_Bin3 - (TIME_TO_REAL(Bin3_Timer.ET) / 1000.0) * Sim_Rate_Bin3;
    ELSE
        Bin3_Timer(IN := FALSE);
    END_IF;
    
    IF Discharge_Bin2 THEN
        Bin2_Timer(IN := TRUE, PT := T#1000S);
        Current_Weight_Bin2 := Start_Weight_Bin2 - (TIME_TO_REAL(Bin2_Timer.ET) / 1000.0) * Sim_Rate_Bin2;
    ELSE
        Bin2_Timer(IN := FALSE);
    END_IF;
    
    IF Discharge_Bin1 THEN
        Bin1_Timer(IN := TRUE, PT := T#1000S);
        Current_Weight_Bin1 := Start_Weight_Bin1 - (TIME_TO_REAL(Bin1_Timer.ET) / 1000.0) * Sim_Rate_Bin1;
    ELSE
        Bin1_Timer(IN := FALSE);
    END_IF;
ELSE
    (* ================= PHYSICAL MODBUS RTU DATA ACQUISITION ================= *)
    (* Uncomment these blocks and their declarations when deploying to physical hardware *)
    (*
    Read_LC1(
        EN := TRUE,
        COM := 1,
        SLV := 1,
        FCT := 3,
        ADDR := 40001,
        SZ := 2,
        DATA := ADR(LC1_Buffer)
    );
    Current_Weight_Bin1 := WORD_TO_REAL(LC1_Buffer[0]);
    
    Read_LC2(
        EN := TRUE,
        COM := 1,
        SLV := 2,
        FCT := 3,
        ADDR := 40001,
        SZ := 2,
        DATA := ADR(LC2_Buffer)
    );
    Current_Weight_Bin2 := WORD_TO_REAL(LC2_Buffer[0]);
    
    Read_LC3(
        EN := TRUE,
        COM := 1,
        SLV := 3,
        FCT := 3,
        ADDR := 40001,
        SZ := 2,
        DATA := ADR(LC3_Buffer)
    );
    Current_Weight_Bin3 := WORD_TO_REAL(LC3_Buffer[0]);
    *)
END_IF;


(* 2. EMERGENCY STOP LOGIC *)
IF E_Stop_Active THEN
    Discharge_Bin1 := FALSE;
    Discharge_Bin2 := FALSE;
    Discharge_Bin3 := FALSE;
    Sequence_Complete := FALSE;
    Step := 0;
    Transition_Timer(IN := FALSE);
    RETURN;
END_IF;


(* 3. SEQUENCE CONTROL *)
IF Auto_Mode THEN
    (* ================= AUTOMATIC MODE ================= *)
    CASE Step OF
        0: (* Idle state *)
            Discharge_Bin1 := FALSE;
            Discharge_Bin2 := FALSE;
            Discharge_Bin3 := FALSE;
            Sequence_Complete := FALSE;
            Transition_Timer(IN := FALSE);
            
            IF Start_Button THEN
                (* Take snapshot of initial load cell weights *)
                Start_Weight_Bin1 := Current_Weight_Bin1;
                Start_Weight_Bin2 := Current_Weight_Bin2;
                Start_Weight_Bin3 := Current_Weight_Bin3;
                
                (* Calculate required cutoff weights based on discharge thresholds *)
                Cutoff_Weight_Bin3 := Start_Weight_Bin3 - Target_Amount_Bin3;
                Cutoff_Weight_Bin2 := Start_Weight_Bin2 - Target_Amount_Bin2;
                Cutoff_Weight_Bin1 := Start_Weight_Bin1 - Target_Amount_Bin1;
                
                Step := 10;
            END_IF
            
        10: (* Discharge Bin 3 - ON *)
            Discharge_Bin3 := TRUE;
            Discharge_Bin2 := FALSE;
            Discharge_Bin1 := FALSE;
            
            (* Check if current weight has dropped below target cutoff *)
            IF Current_Weight_Bin3 <= Cutoff_Weight_Bin3 THEN
                Step := 15;
            END_IF
            
        15: (* Discharge Bin 3 - OFF & Wait Transition Delay *)
            Discharge_Bin3 := FALSE;
            Transition_Timer(IN := TRUE, PT := Step_Delay_Time);
            
            IF Transition_Timer.Q AND (NOT Discharge_Bin3_Feedback OR NOT Discharge_Bin3) THEN
                Transition_Timer(IN := FALSE);
                Step := 20;
            END_IF
            
        20: (* Discharge Bin 2 - ON *)
            Discharge_Bin2 := TRUE;
            Discharge_Bin3 := FALSE;
            Discharge_Bin1 := FALSE;
            
            (* Check if current weight has dropped below target cutoff *)
            IF Current_Weight_Bin2 <= Cutoff_Weight_Bin2 THEN
                Step := 25;
            END_IF
            
        25: (* Discharge Bin 2 - OFF & Wait Transition Delay *)
            Discharge_Bin2 := FALSE;
            Transition_Timer(IN := TRUE, PT := Step_Delay_Time);
            
            IF Transition_Timer.Q AND (NOT Discharge_Bin2_Feedback OR NOT Discharge_Bin2) THEN
                Transition_Timer(IN := FALSE);
                Step := 30;
            END_IF
            
        30: (* Discharge Bin 1 - ON *)
            Discharge_Bin1 := TRUE;
            Discharge_Bin3 := FALSE;
            Discharge_Bin2 := FALSE;
            
            (* Check if current weight has dropped below target cutoff *)
            IF Current_Weight_Bin1 <= Cutoff_Weight_Bin1 THEN
                Step := 35;
            END_IF
            
        35: (* Discharge Bin 1 - OFF & Wait Transition Delay *)
            Discharge_Bin1 := FALSE;
            Transition_Timer(IN := TRUE, PT := Step_Delay_Time);
            
            IF Transition_Timer.Q AND (NOT Discharge_Bin1_Feedback OR NOT Discharge_Bin1) THEN
                Transition_Timer(IN := FALSE);
                Step := 40;
            END_IF
            
        40: (* Sequence Complete *)
            Sequence_Complete := TRUE;
            IF NOT Start_Button THEN
                Step := 0;
            END_IF
    END_CASE;

ELSE
    (* ================= MANUAL MODE ================= *)
    Step := 0;
    Sequence_Complete := FALSE;
    Transition_Timer(IN := FALSE);
    
    (* Separate manual buttons with basic interlinking *)
    IF Manual_Bin3 THEN
        Discharge_Bin3 := TRUE;
        Discharge_Bin2 := FALSE;
        Discharge_Bin1 := FALSE;
    ELSIF Manual_Bin2 THEN
        Discharge_Bin3 := FALSE;
        Discharge_Bin2 := TRUE;
        Discharge_Bin1 := FALSE;
    ELSIF Manual_Bin1 THEN
        Discharge_Bin3 := FALSE;
        Discharge_Bin2 := FALSE;
        Discharge_Bin1 := TRUE;
    ELSE
        Discharge_Bin3 := FALSE;
        Discharge_Bin2 := FALSE;
        Discharge_Bin1 := FALSE;
    END_IF;
END_IF;

END_PROGRAM

// PLC_AC500_V3/Application/batching3
PROGRAM batching3
VAR
    Step : INT := 0;          // Current active step (0: Idle, 1..6: Bins, 7: Delay, 8: Reset & Complete)
    
    (* Mode Control & Commands *)
    Start_Button : BOOL;      // Toggles process start
    E_Stop_Active : BOOL;     // Emergency Stop active signal
    
    (* Cumulative Weighing Variables *)
    load_cell_value : REAL;   // Current weight read from the single load cell
    bin_last_weight : REAL;   // Cumulative baseline weight on the load cell before starting current bin
    actual_bin : REAL;        // Current weight added from active bin
    target_act_bin : REAL;    // Target weight to add from the active bin
    bin_set_value : REAL;     // Setpoint weight for current active step
    
    (* Outputs *)
    Discharge_Bin : ARRAY[1..6] OF BOOL;
    Discharge_Bin_Feedback : ARRAY[1..6] OF BOOL;
    Actual_Weights : ARRAY[1..6] OF REAL; // Actual weight poured per silo
    Sequence_Complete : BOOL;
    
    (* RECIPE DATA STRUCTURES *)
    (* Set Weights array for 20 materials *)
    Recipe_Weights : ARRAY[1..20] OF REAL := [
        50.0,   // Material index 1 target (50.0 kg)
        15.0,   // Material index 2 target (15.0 kg)
        28.0,   // Material index 3 target (28.0 kg)
        31.0,   // Material index 4 target (31.0 kg)
        150.0,  // Material index 5 target (150.0 kg)
        10.0,   // Material index 6 target (10.0 kg)
        0.0, 0.0, 0.0, 0.0, 0.0, 0.0, 0.0, 0.0, 0.0, 0.0, 0.0, 0.0, 0.0, 0.0
    ];
    
    (* Bin Mapping for 6 Bins *)
    (* Contains 1-based Material ID index from Recipe_Weights *)
    (* If 0, the bin is skipped *)
    Bin_Material_Index : ARRAY[1..6] OF INT := [
        1,   // Bin 1 maps to Material 1 (50.0 kg)
        2,   // Bin 2 maps to Material 2 (15.0 kg)
        0,   // Bin 3 is 0 (SKIPPED)
        4,   // Bin 4 maps to Material 4 (31.0 kg)
        5,   // Bin 5 maps to Material 5 (150.0 kg)
        6    // Bin 6 maps to Material 6 (10.0 kg)
    ];
    
    Mat_Idx : INT;            // Active Material Index for lookup
    i : INT;                  // Loop index
    
    (* TIMERS FOR TRANSITIONS & DELAYS *)
    Transition_Timer : TON;
    Completion_Timer : TON;
    Step_Delay_Time : TIME := T#2S;     // Delay between closing one valve and opening the next
    Post_Complete_Delay : TIME := T#2S; // Delay after last bin closes before resetting bin_last_weight
    
    (* SELF-CONTAINED SIMULATION VARIABLES *)
    Simulation_Mode : BOOL := TRUE;
    Sim_Rate : REAL := 10.0;            // Simulated pouring speed (10.0 kg/s)
    Sim_Timer : TON;
    Start_Sim_Weight : REAL;
    Discharge_Active : BOOL;
END_VAR

(* Single Load Cell Cumulative Weighing Sequence (6 Bins with Material Mapping, Skipping, and Self-Contained Simulation) *)

(* 1. SELF-CONTAINED SIMULATION WEIGHT MANAGEMENT *)
IF Simulation_Mode THEN
    (* Reset simulation to baseline (e.g. 2.0 kg) *)
    IF Step = 0 AND NOT Start_Button AND NOT Sequence_Complete THEN
        load_cell_value := 2.0;
        bin_last_weight := 2.0;
        Start_Sim_Weight := 2.0;
        Sim_Timer(IN := FALSE);
    END_IF;
    
    (* Check if any valve is actively discharging *)
    Discharge_Active := FALSE;
    IF Step >= 1 AND Step <= 6 THEN
        Discharge_Active := Discharge_Bin[Step];
    END_IF;
    
    (* Simulate weight gain on the load cell *)
    IF Discharge_Active THEN
        Sim_Timer(IN := TRUE, PT := T#1000S);
        load_cell_value := Start_Sim_Weight + (TIME_TO_REAL(Sim_Timer.ET) / 1000.0) * Sim_Rate;
    ELSE
        Sim_Timer(IN := FALSE);
        Start_Sim_Weight := load_cell_value;
    END_IF;
END_IF;


(* 2. EMERGENCY STOP LOGIC *)
IF E_Stop_Active THEN
    FOR i := 1 TO 6 DO
        Discharge_Bin[i] := FALSE;
        Actual_Weights[i] := 0.0;
    END_FOR;
    Sequence_Complete := FALSE;
    Step := 0;
    Transition_Timer(IN := FALSE);
    Completion_Timer(IN := FALSE);
    RETURN;
END_IF;


(* 3. RECIPE START INITIALIZATION *)
IF Step = 0 AND Start_Button THEN
    Step := 1;
    bin_last_weight := load_cell_value;
    Sequence_Complete := FALSE;
    (* Clear actual weights on start *)
    FOR i := 1 TO 6 DO
        Actual_Weights[i] := 0.0;
    END_FOR;
END_IF;


(* 4. SEQUENCE CONTROL STATE MACHINE *)
CASE Step OF
    1..6: (* Discharging Silos 1 to 6 *)
        Mat_Idx := Bin_Material_Index[Step];
        
        IF Mat_Idx = 0 THEN
            (* Skip this bin instantly and step to next *)
            Step := Step + 1;
        ELSE
            (* Fetch target weight from Recipe_Weights using the mapped material index *)
            bin_set_value := Recipe_Weights[Mat_Idx];
            target_act_bin := bin_set_value;
            
            (* Calculate weight added by current active bin (increasing weight logic) *)
            actual_bin := load_cell_value - bin_last_weight;
            
            (* Update the actual weight in the array for the active bin *)
            Actual_Weights[Step] := actual_bin;
            
            (* Open discharge output valve *)
            Discharge_Bin[Step] := TRUE;
            
            (* Check if target weight has been achieved *)
            IF actual_bin >= target_act_bin THEN
                Discharge_Bin[Step] := FALSE;
                
                (* Set new baseline for the next step *)
                bin_last_weight := load_cell_value;
                
                (* Go to transition delay *)
                Step := 10 + Step; // Offset to separate transition states
            END_IF;
        END_IF;

    11..15: (* Transition Delays (Between Bins) *)
        Transition_Timer(IN := TRUE, PT := Step_Delay_Time);
        IF Transition_Timer.Q AND (NOT Discharge_Bin[Step - 10] OR NOT Discharge_Bin_Feedback[Step - 10]) THEN
            Transition_Timer(IN := FALSE);
            Step := (Step - 10) + 1; // Advance to next bin
        END_IF;
        
    16: (* Transition Delay After Last Bin (Bin 6) Closes *)
        Transition_Timer(IN := TRUE, PT := Step_Delay_Time);
        IF Transition_Timer.Q AND (NOT Discharge_Bin[6] OR NOT Discharge_Bin_Feedback[6]) THEN
            Transition_Timer(IN := FALSE);
            Step := 7; // Go to post-discharge wait step
        END_IF;

    7: (* Wait 2 Seconds After Closing the Last Bin *)
        Completion_Timer(IN := TRUE, PT := Post_Complete_Delay);
        IF Completion_Timer.Q THEN
            Completion_Timer(IN := FALSE);
            Step := 8; // Proceed to reset last weight
        END_IF;
        
    8: (* Reset bin_last_weight to 0 & Complete *)
        bin_last_weight := 0.0;
        Sequence_Complete := TRUE;
        
        IF NOT Start_Button THEN
            Step := 0;
            Sequence_Complete := FALSE;
            (* Reset all actual weights at completion once start is released *)
            FOR i := 1 TO 6 DO
                Actual_Weights[i] := 0.0;
            END_FOR;
        END_IF;
END_CASE;

END_PROGRAM

// PLC_AC500_V3/Application/batching4
PROGRAM batching4
VAR
    Step : INT := 0;          // Current active step (0: Idle, 1..6: Bins, 7: Delay, 8: Reset & Complete)
    
    (* Mode Control & Commands *)
    Start_Button : BOOL;      // Toggles process start
    E_Stop_Active : BOOL;     // Emergency Stop active signal
    
    (* Cumulative Weighing Variables *)
    load_cell_value : REAL;   // Current weight read from the single load cell
    bin_last_weight : REAL;   // Cumulative baseline weight on the load cell before starting current bin
    actual_bin : REAL;        // Current weight added from active bin
    target_act_bin : REAL;    // Target weight to add from the active bin
    bin_set_value : REAL;     // Setpoint weight for current active step
    
    (* Outputs *)
    Discharge_Bin : ARRAY[1..6] OF BOOL;
    Discharge_Bin_Feedback : ARRAY[1..6] OF BOOL;
    Actual_Weights : ARRAY[1..6] OF REAL; // Actual weight poured per silo
    Sequence_Complete : BOOL;
    
    (* RECIPE DATA STRUCTURES *)
    (* Set Weights array for 20 materials *)
    Recipe_Weights : ARRAY[1..20] OF REAL := [
        50.0,   // Material index 1 target (50.0 kg)
        15.0,   // Material index 2 target (15.0 kg)
        28.0,   // Material index 3 target (28.0 kg)
        31.0,   // Material index 4 target (31.0 kg)
        150.0,  // Material index 5 target (150.0 kg)
        10.0,   // Material index 6 target (10.0 kg)
        0.0, 0.0, 0.0, 0.0, 0.0, 0.0, 0.0, 0.0, 0.0, 0.0, 0.0, 0.0, 0.0, 0.0
    ];
    
    (* Bin Mapping for 6 Bins *)
    (* Contains 1-based Material ID index from Recipe_Weights *)
    (* If 0, the bin is skipped *)
    Bin_Material_Index : ARRAY[1..6] OF INT := [
        1,   // Bin 1 maps to Material 1 (50.0 kg)
        2,   // Bin 2 maps to Material 2 (15.0 kg)
        0,   // Bin 3 is 0 (SKIPPED)
        4,   // Bin 4 maps to Material 4 (31.0 kg)
        5,   // Bin 5 maps to Material 5 (150.0 kg)
        6    // Bin 6 maps to Material 6 (10.0 kg)
    ];
    
    Mat_Idx : INT;            // Active Material Index for lookup
    i : INT;                  // Loop index
    
    (* TIMERS FOR TRANSITIONS & DELAYS *)
    Transition_Timer : TON;
    Completion_Timer : TON;
    Step_Delay_Time : TIME := T#2S;     // Delay between closing one valve and opening the next
    Post_Complete_Delay : TIME := T#2S; // Delay after last bin closes before resetting bin_last_weight
    
    (* SELF-CONTAINED SIMULATION VARIABLES *)
    Simulation_Mode : BOOL := TRUE;
    Sim_Rate : REAL := 10.0;            // Simulated pouring speed (10.0 kg/s)
    Sim_Timer : TON;
    Start_Sim_Weight : REAL;
    Discharge_Active : BOOL;
END_VAR

(* Single Load Cell Cumulative Weighing Sequence (6 Bins with Material Mapping, Skipping, and Self-Contained Simulation) *)

(* 1. SELF-CONTAINED SIMULATION WEIGHT MANAGEMENT *)
IF Simulation_Mode THEN
    (* Reset simulation to baseline (e.g. 2.0 kg) *)
    IF Step = 0 AND NOT Start_Button AND NOT Sequence_Complete THEN
        load_cell_value := 0.0;
        bin_last_weight := 0.0;
        Start_Sim_Weight := 0.0;
        Sim_Timer(IN := FALSE);
    END_IF;
    
    (* Check if any valve is actively discharging *)
    Discharge_Active := FALSE;
    IF Step >= 1 AND Step <= 6 THEN
        Discharge_Active := Discharge_Bin[Step];
    END_IF;
    
    (* Simulate weight gain on the load cell *)
    IF Discharge_Active THEN
        Sim_Timer(IN := TRUE, PT := T#1000S);
        load_cell_value := Start_Sim_Weight + (TIME_TO_REAL(Sim_Timer.ET) / 1000.0) * Sim_Rate;
    ELSE
        Sim_Timer(IN := FALSE);
        Start_Sim_Weight := load_cell_value;
    END_IF;
END_IF;


(* 2. EMERGENCY STOP LOGIC *)
IF E_Stop_Active THEN
    FOR i := 1 TO 6 DO
        Discharge_Bin[i] := FALSE;
        Actual_Weights[i] := 0.0;
    END_FOR;
    Sequence_Complete := FALSE;
    Step := 0;
    Transition_Timer(IN := FALSE);
    Completion_Timer(IN := FALSE);
    RETURN;
END_IF;


(* 3. RECIPE START INITIALIZATION *)
IF Step = 0 AND Start_Button THEN
    Step := 1;
    bin_last_weight := load_cell_value;
    Sequence_Complete := FALSE;
    (* Clear actual weights on start *)
    FOR i := 1 TO 6 DO
        Actual_Weights[i] := 0.0;
    END_FOR;
END_IF;


(* 4. SEQUENCE CONTROL STATE MACHINE *)
CASE Step OF
    1..6: (* Discharging Silos 1 to 6 *)
        Mat_Idx := Bin_Material_Index[Step];
        
        IF Mat_Idx = 0 THEN
            (* Skip this bin instantly and step to next *)
            Step := Step + 1;
        ELSE
            (* Fetch target weight from Recipe_Weights using the mapped material index *)
            bin_set_value := Recipe_Weights[Mat_Idx];
            target_act_bin := bin_set_value;
            
            (* Calculate weight added by current active bin (increasing weight logic) *)
            actual_bin := load_cell_value - bin_last_weight;
            
            (* Update the actual weight in the array for the active bin *)
            Actual_Weights[Step] := actual_bin;
            
            (* Open discharge output valve *)
            Discharge_Bin[Step] := TRUE;
            
            (* Check if target weight has been achieved *)
            IF actual_bin >= target_act_bin THEN
                Discharge_Bin[Step] := FALSE;
                
                (* Set new baseline for the next step *)
                bin_last_weight := load_cell_value;
                
                (* Go to transition delay *)
                Step := 10 + Step; // Offset to separate transition states
            END_IF;
        END_IF;

    11..15: (* Transition Delays (Between Bins) *)
        Transition_Timer(IN := TRUE, PT := Step_Delay_Time);
        IF Transition_Timer.Q AND (NOT Discharge_Bin[Step - 10] OR NOT Discharge_Bin_Feedback[Step - 10]) THEN
            Transition_Timer(IN := FALSE);
            Step := (Step - 10) + 1; // Advance to next bin
        END_IF;
        
    16: (* Transition Delay After Last Bin (Bin 6) Closes *)
        Transition_Timer(IN := TRUE, PT := Step_Delay_Time);
        IF Transition_Timer.Q AND (NOT Discharge_Bin[6] OR NOT Discharge_Bin_Feedback[6]) THEN
            Transition_Timer(IN := FALSE);
            Step := 7; // Go to post-discharge wait step
        END_IF;

    7: (* Wait 2 Seconds After Closing the Last Bin *)
        Completion_Timer(IN := TRUE, PT := Post_Complete_Delay);
        IF Completion_Timer.Q THEN
            Completion_Timer(IN := FALSE);
            Step := 8; // Proceed to reset last weight
        END_IF;
        
    8: (* Reset bin_last_weight & Complete *)
    bin_last_weight := 0.0;
    Sequence_Complete := TRUE;

    (* Reset all actual weights *)
    FOR i := 1 TO 6 DO
        Actual_Weights[i] := 0.0;
    END_FOR;

    IF NOT Start_Button THEN
        Step := 0;
        Sequence_Complete := FALSE;
    END_IF;
END_CASE;

END_PROGRAM

// PLC_AC500_V3/Application/batching5
PROGRAM batching5
VAR
    Step : INT := 0;          // Current active step (0: Idle, 1..6: Bins, 7: Delay, 8: Reset & Complete)
    
    (* Mode Control & Commands *)
    Start_Button : BOOL;      // Toggles process start
    E_Stop_Active : BOOL;     // Emergency Stop active signal
    
    (* Cumulative Weighing Variables *)
    load_cell_value : REAL;   // Current weight read from the single load cell
    bin_last_weight : REAL;   // Cumulative baseline weight on the load cell before starting current bin
    actual_bin : REAL;        // Current weight added from active bin
    target_act_bin : REAL;    // Target weight to add from the active bin
    bin_set_value : REAL;     // Setpoint weight for current active step
    slow_cutoff_weight : REAL; // Cutoff threshold weight to switch from FAST to SLOW feed
    
    (* Dynamic Display Text *)
    Status_Message : STRING := 'System Idle';
    
    (* Outputs *)
    Discharge_Bin_Coarse : ARRAY[1..6] OF BOOL; // Coarse feed valve outputs
    Discharge_Bin_Fine : ARRAY[1..6] OF BOOL;   // Fine feed valve outputs
    Discharge_Bin_Feedback : ARRAY[1..6] OF BOOL;
    Actual_Weights : ARRAY[1..6] OF REAL; // Actual weight poured per silo
    Sequence_Complete : BOOL;
    
    (* RECIPE DATA STRUCTURES *)
    (* Set Weights array for 20 materials *)
    Recipe_Weights : ARRAY[1..20] OF REAL := [
        50.0,   // Material index 1 target (50.0 kg)
        15.0,   // Material index 2 target (15.0 kg)
        28.0,   // Material index 3 target (28.0 kg)
        31.0,   // Material index 4 target (31.0 kg)
        150.0,  // Material index 5 target (150.0 kg)
        10.0,   // Material index 6 target (10.0 kg)
        0.0, 0.0, 0.0, 0.0, 0.0, 0.0, 0.0, 0.0, 0.0, 0.0, 0.0, 0.0, 0.0, 0.0
    ];
    
    (* Set Slow Feed Transition Percentages for 20 materials *)
    (* E.g., 20.0 = Slow down when 20% of target weight is remaining *)
    Recipe_Slow_Pcts : ARRAY[1..20] OF REAL := [
        20.0,   // Silo 1: Slow down at 80% (40.0 kg)
        20.0,   // Silo 2: Slow down at 80% (12.0 kg)
        20.0,   // Silo 3: Slow down at 80%
        20.0,   // Silo 4: Slow down at 80%
        20.0,   // Silo 5: Slow down at 80%
        20.0,   // Silo 6: Slow down at 80% (8.0 kg)
        0.0, 0.0, 0.0, 0.0, 0.0, 0.0, 0.0, 0.0, 0.0, 0.0, 0.0, 0.0, 0.0, 0.0
    ];
    
    (* Bin Mapping for 6 Bins *)
    (* Contains 1-based Material ID index from Recipe_Weights *)
    (* If 0, the bin is skipped *)
    Bin_Material_Index : ARRAY[1..6] OF INT := [
        1,   // Bin 1 maps to Material 1 (50.0 kg)
        2,   // Bin 2 maps to Material 2 (15.0 kg)
        0,   // Bin 3 is 0 (SKIPPED)
        4,   // Bin 4 maps to Material 4 (31.0 kg)
        5,   // Bin 5 maps to Material 5 (150.0 kg)
        6    // Bin 6 maps to Material 6 (10.0 kg)
    ];
    
    Mat_Idx : INT;            // Active Material Index for lookup
    i : INT;                  // Loop index
    
    (* TIMERS FOR TRANSITIONS & DELAYS *)
    Transition_Timer : TON;
    Completion_Timer : TON;
    Step_Delay_Time : TIME := T#2S;     // Delay between closing one valve and opening the next
    Post_Complete_Delay : TIME := T#2S; // Delay after last bin closes before resetting bin_last_weight
    
    (* SELF-CONTAINED SIMULATION VARIABLES *)
    Simulation_Mode : BOOL := TRUE;
    Sim_Rate : REAL := 10.0;            // Simulated pouring speed (10.0 kg/s during fast feed)
    Sim_Timer : TON;
    Start_Sim_Weight : REAL;
    Discharge_Active : BOOL;
END_VAR

(* Single Load Cell Cumulative Weighing Sequence (6 Bins with Mutually Exclusive Speed Transition and Tolerance Message) *)

(* 1. SELF-CONTAINED SIMULATION WEIGHT MANAGEMENT *)
IF Simulation_Mode THEN
    (* Reset simulation to baseline (e.g. 2.0 kg) *)
    IF Step = 0 AND NOT Start_Button AND NOT Sequence_Complete THEN
        load_cell_value := 2.0;
        bin_last_weight := 2.0;
        Start_Sim_Weight := 2.0;
        Sim_Timer(IN := FALSE);
    END_IF;
    
    (* Check if any valve is actively discharging (either Coarse or Fine) *)
    Discharge_Active := FALSE;
    IF Step >= 1 AND Step <= 6 THEN
        Discharge_Active := Discharge_Bin_Coarse[Step] OR Discharge_Bin_Fine[Step];
    END_IF;
    
    (* Simulate weight gain on the load cell *)
    IF Discharge_Active THEN
        Sim_Timer(IN := TRUE, PT := T#1000S);
        load_cell_value := Start_Sim_Weight + (TIME_TO_REAL(Sim_Timer.ET) / 1000.0) * Sim_Rate;
    ELSE
        Sim_Timer(IN := FALSE);
        Start_Sim_Weight := load_cell_value;
    END_IF;
END_IF;


(* 2. EMERGENCY STOP LOGIC *)
IF E_Stop_Active THEN
    FOR i := 1 TO 6 DO
        Discharge_Bin_Coarse[i] := FALSE;
        Discharge_Bin_Fine[i] := FALSE;
        Actual_Weights[i] := 0.0;
    END_FOR;
    Sequence_Complete := FALSE;
    Step := 0;
    Status_Message := 'E-Stop Active!';
    Transition_Timer(IN := FALSE);
    Completion_Timer(IN := FALSE);
    RETURN;
END_IF;


(* 3. RECIPE START INITIALIZATION *)
IF Step = 0 AND Start_Button THEN
    Step := 1;
    bin_last_weight := load_cell_value;
    Sequence_Complete := FALSE;
    Status_Message := 'Batch Started';
    (* Clear actual weights on start *)
    FOR i := 1 TO 6 DO
        Actual_Weights[i] := 0.0;
    END_FOR;
END_IF;


(* 4. SEQUENCE CONTROL STATE MACHINE *)
CASE Step OF
    1..6: (* Discharging Silos 1 to 6 *)
        Mat_Idx := Bin_Material_Index[Step];
        
        IF Mat_Idx = 0 THEN
            (* Skip this bin instantly and step to next *)
            Step := Step + 1;
        ELSE
            (* Fetch target weight from Recipe_Weights using the mapped material index *)
            bin_set_value := Recipe_Weights[Mat_Idx];
            target_act_bin := bin_set_value;
            
            (* Calculate slow-down cutoff weight (e.g. 20% of target left) *)
            slow_cutoff_weight := target_act_bin - (target_act_bin * (Recipe_Slow_Pcts[Mat_Idx] / 100.0));
            
            (* Calculate weight added by current active bin (increasing weight logic) *)
            actual_bin := load_cell_value - bin_last_weight;
            
            (* Update the actual weight in the array for the active bin *)
            Actual_Weights[Step] := actual_bin;
            
            (* Dual-Speed Output Control & Simulation Rate Scaling *)
            IF actual_bin < slow_cutoff_weight THEN
                Discharge_Bin_Coarse[Step] := TRUE;
                Discharge_Bin_Fine[Step] := FALSE; // Mutual Exclusivity - Coarse ONLY
                Status_Message := 'Fast feeding active';
                Sim_Rate := 10.0; // Fast simulation rate
            ELSE
                Discharge_Bin_Coarse[Step] := FALSE; // Shut off coarse motor
                Discharge_Bin_Fine[Step] := TRUE;  // Mutual Exclusivity - Fine ONLY
                Status_Message := 'Tolerance weight is going on so motor is slow';
                Sim_Rate := 2.0;  // Slow simulation rate
            END_IF;
            
            (* Check if target weight has been achieved *)
            IF actual_bin >= target_act_bin THEN
                Discharge_Bin_Coarse[Step] := FALSE;
                Discharge_Bin_Fine[Step] := FALSE;
                
                (* Set new baseline for the next step *)
                bin_last_weight := load_cell_value;
                Status_Message := 'Bin Step Completed';
                
                (* Go to transition delay *)
                Step := 10 + Step; // Offset to separate transition states
            END_IF;
        END_IF;

    11..15: (* Transition Delays (Between Bins) *)
        Transition_Timer(IN := TRUE, PT := Step_Delay_Time);
        (* Verify both coarse and fine outputs are off, and feedback conforms *)
        IF Transition_Timer.Q AND (NOT Discharge_Bin_Coarse[Step - 10] AND NOT Discharge_Bin_Fine[Step - 10]) THEN
            Transition_Timer(IN := FALSE);
            Step := (Step - 10) + 1; // Advance to next bin
        END_IF;
        
    16: (* Transition Delay After Last Bin (Bin 6) Closes *)
        Transition_Timer(IN := TRUE, PT := Step_Delay_Time);
        IF Transition_Timer.Q AND (NOT Discharge_Bin_Coarse[6] AND NOT Discharge_Bin_Fine[6]) THEN
            Transition_Timer(IN := FALSE);
            Step := 7; // Go to post-discharge wait step
        END_IF;

    7: (* Wait 2 Seconds After Closing the Last Bin *)
        Status_Message := 'Settling delay active';
        Completion_Timer(IN := TRUE, PT := Post_Complete_Delay);
        IF Completion_Timer.Q THEN
            Completion_Timer(IN := FALSE);
            Step := 8; // Proceed to reset last weight
        END_IF;
        
    8: (* Reset bin_last_weight to 0 & Complete *)
        bin_last_weight := 0.0;
        Sequence_Complete := TRUE;
        Status_Message := 'Sequence Completed';
        
        IF NOT Start_Button THEN
            Step := 0;
            Sequence_Complete := FALSE;
            Status_Message := 'System Idle';
            (* Reset all actual weights at completion once start is released *)
            FOR i := 1 TO 6 DO
                Actual_Weights[i] := 0.0;
            END_FOR;
        END_IF;
END_CASE;

END_PROGRAM

// PLC_AC500_V3/Application/Auto_Batching
FUNCTION_BLOCK Auto_Batching
VAR_INPUT
    Start_Button : BOOL;      // Signal to start the batching sequence
    E_Stop_Active : BOOL;     // Emergency Stop active signal
    load_cell_value : REAL;   // Weight value read from load cell
    Discharge_Bin_Feedback : ARRAY[1..6] OF BOOL; // Physical valve feedbacks
END_VAR
VAR_OUTPUT
    Auto_Bin : ARRAY[1..6] OF BOOL; // Motor/valve control outputs
    Actual_Weights : ARRAY[1..6] OF REAL; // Actual weight poured per silo
    Sequence_Complete : BOOL;  // Batch complete flag
END_VAR
VAR
    Step : INT := 0;          // State machine index (0: Idle, 1..6: Bins, 7: Delay, 8: Reset)
    bin_last_weight : REAL;   // Baseline weight on the load cell before starting current bin
    actual_bin : REAL;        // Current weight added from active bin
    target_act_bin : REAL;    // Target weight to add from the active bin
    bin_set_value : REAL;     // Setpoint weight for current active step
    
    (* Bin Mapping for 6 Auto Bins *)
    (* Maps physical Silo 1..6 to Material Index 1..20 *)
    Bin_Material_Index : ARRAY[1..6] OF INT := [
        1,   // Bin 1 maps to Material 1 (50.0 kg)
        2,   // Bin 2 maps to Material 2 (15.0 kg)
        0,   // Bin 3 is 0 (SKIPPED)
        4,   // Bin 4 maps to Material 4 (31.0 kg)
        5,   // Bin 5 maps to Material 5 (150.0 kg)
        6    // Bin 6 maps to Material 6 (10.0 kg)
    ];
    
    Mat_Idx : INT;
    i : INT;                  // General loop index
    
    (* TIMERS FOR TRANSITIONS & DELAYS *)
    Transition_Timer : TON;
    Completion_Timer : TON;
    Step_Delay_Time : TIME := T#2S;
    Post_Complete_Delay : TIME := T#2S;
    
    (* SELF-CONTAINED SIMULATION VARIABLES *)
    Simulation_Mode : BOOL := TRUE;
    Sim_Rate : REAL := 10.0;            // Simulated pouring speed (10.0 kg/s)
    Sim_Timer : TON;
    Start_Sim_Weight : REAL;
    Discharge_Active : BOOL;
END_VAR

(* Cumulative Gain-in-Weight Auto Batching FB *)

(* 1. SELF-CONTAINED SIMULATION WEIGHT MANAGEMENT *)
IF Simulation_Mode THEN
    (* Reset simulation to baseline (e.g. 2.0 kg) *)
    IF Step = 0 AND NOT Start_Button AND NOT Sequence_Complete THEN
        load_cell_value := 2.0;
        bin_last_weight := 2.0;
        Start_Sim_Weight := 2.0;
        Sim_Timer(IN := FALSE);
    END_IF;
    
    (* Check if any valve is actively discharging *)
    Discharge_Active := FALSE;
    IF Step >= 1 AND Step <= 6 THEN
        Discharge_Active := Auto_Bin[Step];
    END_IF;
    
    (* Simulate weight gain on the load cell *)
    IF Discharge_Active THEN
        Sim_Timer(IN := TRUE, PT := T#1000S);
        load_cell_value := Start_Sim_Weight + (TIME_TO_REAL(Sim_Timer.ET) / 1000.0) * Sim_Rate;
    ELSE
        Sim_Timer(IN := FALSE);
        Start_Sim_Weight := load_cell_value;
    END_IF;
END_IF;


(* 2. EMERGENCY STOP LOGIC *)
IF E_Stop_Active THEN
    FOR i := 1 TO 6 DO
        Auto_Bin[i] := FALSE;
        Actual_Weights[i] := 0.0;
    END_FOR;
    Sequence_Complete := FALSE;
    Step := 0;
    Transition_Timer(IN := FALSE);
    Completion_Timer(IN := FALSE);
    RETURN;
END_IF;


(* 3. RECIPE SEQUENCE START *)
IF Step = 0 AND Start_Button THEN
    Step := 1;
    bin_last_weight := load_cell_value;
    Sequence_Complete := FALSE;
    (* Clear actual weights on start *)
    FOR i := 1 TO 6 DO
        Actual_Weights[i] := 0.0;
    END_FOR;
END_IF;


(* 4. SEQUENCE CONTROL STATE MACHINE *)
CASE Step OF
    1..6: (* Discharging Silos 1 to 6 *)
        Mat_Idx := Bin_Material_Index[Step];
        
        IF Mat_Idx = 0 THEN
            (* Skip this bin instantly *)
            Step := Step + 1;
        ELSE
            (* Fetch target weight from global Recipe_Weights array *)
            bin_set_value := GVL.Recipe_Weights[Mat_Idx];
            target_act_bin := bin_set_value;
            
            (* Calculate weight added by current active bin *)
            actual_bin := load_cell_value - bin_last_weight;
            
            (* Update the actual weight in the array for the active bin *)
            Actual_Weights[Step] := actual_bin;
            
            (* Open discharge output valve *)
            Auto_Bin[Step] := TRUE;
            
            (* Check if target weight has been achieved *)
            IF actual_bin >= target_act_bin THEN
                Auto_Bin[Step] := FALSE;
                
                (* Set new baseline for the next step *)
                bin_last_weight := load_cell_value;
                
                (* Go to transition delay *)
                Step := 10 + Step; // Offset to separate transition states
            END_IF;
        END_IF;

    11..15: (* Transition Delays (Between Bins) *)
        Transition_Timer(IN := TRUE, PT := Step_Delay_Time);
        IF Transition_Timer.Q AND (NOT Auto_Bin[Step - 10] OR NOT Discharge_Bin_Feedback[Step - 10]) THEN
            Transition_Timer(IN := FALSE);
            Step := (Step - 10) + 1; // Advance to next bin
        END_IF;
        
    16: (* Transition Delay After Last Bin (Bin 6) Closes *)
        Transition_Timer(IN := TRUE, PT := Step_Delay_Time);
        IF Transition_Timer.Q AND (NOT Auto_Bin[6] OR NOT Discharge_Bin_Feedback[6]) THEN
            Transition_Timer(IN := FALSE);
            Step := 7; // Go to post-discharge wait step
        END_IF;

    7: (* Wait 2 Seconds After Closing the Last Bin *)
        Completion_Timer(IN := TRUE, PT := Post_Complete_Delay);
        IF Completion_Timer.Q THEN
            Completion_Timer(IN := FALSE);
            Step := 8; // Proceed to reset last weight
        END_IF;
        
    8: (* Reset bin_last_weight to 0 & Complete *)
        bin_last_weight := 0.0;
        Sequence_Complete := TRUE;
        
        IF NOT Start_Button THEN
            Step := 0;
            Sequence_Complete := FALSE;
            (* Reset all actual weights at completion once start is released *)
            FOR i := 1 TO 6 DO
                Actual_Weights[i] := 0.0;
            END_FOR;
        END_IF;
END_CASE;

END_FUNCTION_BLOCK

// PLC_AC500_V3/Application/Manual_Batching
FUNCTION_BLOCK Manual_Batching
VAR_INPUT
    Start_Button : BOOL;      // Signal to start the batching sequence
    E_Stop_Active : BOOL;     // Emergency Stop active signal
    load_cell_value : REAL;   // Weight value read from load cell
END_VAR
VAR_OUTPUT
    Manual_Bin : ARRAY[1..10] OF BOOL; // Prompts/indicators for Bins 7..16
    Actual_Weights : ARRAY[1..10] OF REAL; // Actual weight poured per silo
    Sequence_Complete : BOOL;  // Batch complete flag
END_VAR
VAR
    Step : INT := 0;          // State machine index (0: Idle, 1..10: Bins, 11..20: Delays, 30: Settling, 40: Complete)
    bin_last_weight : REAL;   // Baseline weight on the load cell before starting current bin
    actual_bin : REAL;        // Current weight added from active bin
    target_act_bin : REAL;    // Target weight to add from the active bin
    bin_set_value : REAL;     // Setpoint weight for current active step
    
    (* Bin Mapping for 10 Manual Bins *)
    (* Maps physical manual Silo 7..16 to Material Index 1..20 *)
    Bin_Manual_Index : ARRAY[1..10] OF INT := [
        7,    // Silo 7 maps to Material 7 (12.0 kg)
        8,    // Silo 8 maps to Material 8 (8.0 kg)
        0,    // Silo 9 is 0 (SKIPPED)
        10,   // Silo 10 maps to Material 10 (5.0 kg)
        11,   // Silo 11 maps to Material 11 (18.0 kg)
        12,   // Silo 12 maps to Material 12 (22.0 kg)
        13,   // Silo 13 maps to Material 13 (30.0 kg)
        14,   // Silo 14 maps to Material 14 (14.0 kg)
        15,   // Silo 15 maps to Material 15 (9.0 kg)
        16    // Silo 16 maps to Material 16 (11.0 kg)
    ];
    
    Mat_Idx : INT;
    i : INT;                  // General loop index
    
    (* TIMERS FOR TRANSITIONS & DELAYS *)
    Transition_Timer : TON;
    Completion_Timer : TON;
    Step_Delay_Time : TIME := T#2S;
    Post_Complete_Delay : TIME := T#2S;
    
    (* SELF-CONTAINED SIMULATION VARIABLES *)
    Simulation_Mode : BOOL := TRUE;
    Sim_Rate : REAL := 10.0;            // Simulated pouring speed (10.0 kg/s)
    Sim_Timer : TON;
    Start_Sim_Weight : REAL;
    Discharge_Active : BOOL;
END_VAR

(* Cumulative Gain-in-Weight Manual Batching FB (Simulates Operator Pouring) *)

(* 1. SIMULATION WEIGHT MANAGEMENT *)
IF Simulation_Mode THEN
    (* Reset simulation to baseline (e.g. 2.0 kg) *)
    IF Step = 0 AND NOT Start_Button AND NOT Sequence_Complete THEN
        load_cell_value := 2.0;
        bin_last_weight := 2.0;
        Start_Sim_Weight := 2.0;
        Sim_Timer(IN := FALSE);
    END_IF;
    
    (* Check if operator is actively pouring *)
    Discharge_Active := FALSE;
    IF Step >= 1 AND Step <= 10 THEN
        Discharge_Active := Manual_Bin[Step];
    END_IF;
    
    (* Simulate weight gain on the load cell *)
    IF Discharge_Active THEN
        Sim_Timer(IN := TRUE, PT := T#1000S);
        load_cell_value := Start_Sim_Weight + (TIME_TO_REAL(Sim_Timer.ET) / 1000.0) * Sim_Rate;
    ELSE
        Sim_Timer(IN := FALSE);
        Start_Sim_Weight := load_cell_value;
    END_IF;
END_IF;


(* 2. EMERGENCY STOP LOGIC *)
IF E_Stop_Active THEN
    FOR i := 1 TO 10 DO
        Manual_Bin[i] := FALSE;
        Actual_Weights[i] := 0.0;
    END_FOR;
    Sequence_Complete := FALSE;
    Step := 0;
    Transition_Timer(IN := FALSE);
    Completion_Timer(IN := FALSE);
    RETURN;
END_IF;


(* 3. RECIPE SEQUENCE START *)
IF Step = 0 AND Start_Button THEN
    Step := 1;
    bin_last_weight := load_cell_value;
    Sequence_Complete := FALSE;
    (* Clear actual weights on start *)
    FOR i := 1 TO 10 DO
        Actual_Weights[i] := 0.0;
    END_FOR;
END_IF;


(* 4. SEQUENCE CONTROL STATE MACHINE *)
CASE Step OF
    1..10: (* Prompts Silos 7 to 16 *)
        Mat_Idx := Bin_Manual_Index[Step];
        
        IF Mat_Idx = 0 THEN
            (* Skip this bin instantly *)
            Step := Step + 1;
        ELSE
            (* Fetch target weight from global Recipe_Weights array *)
            bin_set_value := GVL.Recipe_Weights[Mat_Idx];
            target_act_bin := bin_set_value;
            
            (* Calculate weight added by current active bin *)
            actual_bin := load_cell_value - bin_last_weight;
            
            (* Update the actual weight in the array for the active bin *)
            Actual_Weights[Step] := actual_bin;
            
            (* Prompt operator indicator active *)
            Manual_Bin[Step] := TRUE;
            
            (* Check if target weight has been achieved *)
            IF actual_bin >= target_act_bin THEN
                Manual_Bin[Step] := FALSE;
                
                (* Set new baseline for the next step *)
                bin_last_weight := load_cell_value;
                
                (* Go to transition delay *)
                Step := 10 + Step; // Offset to separate transition states
            END_IF;
        END_IF;

    11..19: (* Transition Delays (Between Bins) *)
        Transition_Timer(IN := TRUE, PT := Step_Delay_Time);
        IF Transition_Timer.Q THEN
            Transition_Timer(IN := FALSE);
            Step := (Step - 10) + 1; // Advance to next bin
        END_IF;
        
    20: (* Transition Delay After Last Bin (Bin 10) Closes *)
        Transition_Timer(IN := TRUE, PT := Step_Delay_Time);
        IF Transition_Timer.Q THEN
            Transition_Timer(IN := FALSE);
            Step := 30; // Go to post-discharge wait step (State 30)
        END_IF;

    30: (* Wait 2 Seconds After Closing the Last Bin *)
        Completion_Timer(IN := TRUE, PT := Post_Complete_Delay);
        IF Completion_Timer.Q THEN
            Completion_Timer(IN := FALSE);
            Step := 40; // Proceed to reset last weight (State 40)
        END_IF;
        
    40: (* Reset bin_last_weight to 0 & Complete *)
        bin_last_weight := 0.0;
        Sequence_Complete := TRUE;
        
        IF NOT Start_Button THEN
            Step := 0;
            Sequence_Complete := FALSE;
            (* Reset all actual weights at completion once start is released *)
            FOR i := 1 TO 10 DO
                Actual_Weights[i] := 0.0;
            END_FOR;
        END_IF;
END_CASE;

END_FUNCTION_BLOCK

// PLC_AC500_V3/Application/batching6
PROGRAM batching6
VAR
    Auto_Ctrl : Auto_Batching;
    Manual_Ctrl : Manual_Batching;
    
    (* Global Inputs & Toggles *)
    Start_Button : BOOL;
    E_Stop_Active : BOOL;
    
    (* Parallel Weight Feedbacks *)
    load_cell_auto : REAL;
    load_cell_manual : REAL;
    
    (* Process Outputs *)
    Auto_Bin : ARRAY[1..6] OF BOOL;
    Manual_Bin : ARRAY[1..10] OF BOOL;
    
    Auto_Weights : ARRAY[1..6] OF REAL;
    Manual_Weights : ARRAY[1..10] OF REAL;
    
    Auto_Complete : BOOL;
    Manual_Complete : BOOL;
    Sequence_Complete : BOOL;
END_VAR

(* Run Auto & Manual Batching pipelines concurrently in parallel *)

Auto_Ctrl(
    Start_Button := Start_Button,
    E_Stop_Active := E_Stop_Active,
    load_cell_value := load_cell_auto,
    Discharge_Bin_Feedback := ,
    Auto_Bin => Auto_Bin,
    Actual_Weights => Auto_Weights,
    Sequence_Complete => Auto_Complete
);

Manual_Ctrl(
    Start_Button := Start_Button,
    E_Stop_Active := E_Stop_Active,
    load_cell_value := load_cell_manual,
    Manual_Bin => Manual_Bin,
    Actual_Weights => Manual_Weights,
    Sequence_Complete => Manual_Complete
);

(* Global complete once both streams conclude *)
Sequence_Complete := Auto_Complete AND Manual_Complete;

END_PROGRAM

// PLC_AC500_V3/Application/Auto_Batching_V9
FUNCTION_BLOCK Auto_Batching_V9
VAR_INPUT
    Start_Button : BOOL;      // Signal to start the batching sequence
    E_Stop_Active : BOOL;     // Emergency Stop active signal
    Discharge_Bin_Feedback : ARRAY[1..6] OF BOOL; // Physical valve feedbacks
    Auto_Bin_Material_Mapping : ARRAY[1..6] OF INT; // Material index mapping for 6 bins
    Auto_Bin_Cutoff_Weights : ARRAY[1..6] OF REAL; // Cutoff weight thresholds (kg)
    Auto_Bin_Tolerance : ARRAY[1..6] OF REAL; // Tolerance weight offset values (kg)
END_VAR
VAR_IN_OUT
    load_cell_value : REAL;   // Weight value read/written from load cell
END_VAR
VAR_OUTPUT
    Auto_Bin : ARRAY[1..6] OF BOOL; // Coarse feed valve outputs
    auto_bin_cutoff : ARRAY[1..6] OF BOOL; // Fine feed cutoff trigger indicators
    auto_bin_motor : ARRAY[1..6] OF BOOL; // Main conveyor motor outputs
    Actual_Weights : ARRAY[1..6] OF REAL; // Actual weight poured per silo
    Sequence_Complete : BOOL;  // Batch complete flag
    Active_Material_ID : INT;  // Currently active ingredient ID
    Active_Bin_ID : INT;       // Currently active physical Bin ID (1..6)
    Active_Target_Weight : REAL; // Recipe target weight of active bin (with tolerance applied)
    Error_Code : INT;          // Active error code
    Status_Message : STRING;   // Diagnostic text message
END_VAR
VAR
    Step : INT := 0;          // State machine index (0: Idle, 1..6: Bins, 11..16: Delays, 7: Settling, 8: Complete, 99: Error)
    bin_last_weight : REAL;   // Baseline weight on the load cell before starting current bin
    actual_bin : REAL;        // Current weight added from active bin
    target_act_bin : REAL;    // Effective target weight to add from the active bin (GVL target - Tolerance)
    bin_set_value : REAL;     // Setpoint weight looked up from GVL
    cutoff_trigger_weight : REAL; // Calculated trigger weight (target - Tolerance - Cutoff)
    
    Mat_Idx : INT;
    i : INT;                  // General loop index
    
    (* TIMERS FOR TRANSITIONS & DELAYS *)
    Transition_Timer : TON;
    Completion_Timer : TON;
    Step_Delay_Time : TIME := T#2S;
    Post_Complete_Delay : TIME := T#2S;
    
    (* SELF-CONTAINED SIMULATION VARIABLES *)
    Simulation_Mode : BOOL := TRUE;
    Sim_Rate : REAL := 10.0;            // Simulated pouring speed (10.0 kg/s)
    Sim_Timer : TON;
    Start_Sim_Weight : REAL;
    Discharge_Active : BOOL;
END_VAR

(* Auto Batching FB V9 with Tolerance Logic *)

(* 1. SELF-CONTAINED SIMULATION WEIGHT MANAGEMENT *)
IF Simulation_Mode AND Step <> 99 THEN
    (* Reset simulation to baseline *)
    IF Step = 0 AND NOT Start_Button AND NOT Sequence_Complete THEN
        load_cell_value := 0.0;
        bin_last_weight := 0.0;
        Start_Sim_Weight := 0.0;
        Sim_Timer(IN := FALSE);
    END_IF;
    
    (* Check if any valve is actively discharging *)
    Discharge_Active := FALSE;
    IF Step >= 1 AND Step <= 6 THEN
        Discharge_Active := auto_bin_motor[Step];
    END_IF;
    
    (* Simulate weight gain on the load cell *)
    IF Discharge_Active THEN
        Sim_Timer(IN := TRUE, PT := T#1000S);
        load_cell_value := Start_Sim_Weight + (TIME_TO_REAL(Sim_Timer.ET) / 1000.0) * Sim_Rate;
    ELSE
        Sim_Timer(IN := FALSE);
        Start_Sim_Weight := load_cell_value;
    END_IF;
END_IF;


